LIN {X 0,Y 537.383,Z 578.92,A -85,B 0,C 180,E1 13527.001,E2 13527.001} C_VEL
LIN {X 0,Y 529.562,Z 566.226,A -85,B 0,C 180,E1 13524.901,E2 13524.901} C_VEL
LIN {X 0,Y 521.572,Z 553.811,A -85,B 0,C 180,E1 13522.516,E2 13522.516} C_VEL
LIN {X 0,Y 516.394,Z 546.392,A -85,B 0,C 180,E1 13520.813,E2 13520.813} C_VEL
LIN {X 0,Y 512.056,Z 540.726,A -85,B 0,C 180,E1 13519.269,E2 13519.269} C_VEL
LIN {X 0,Y 508.587,Z 536.104,A -85,B 0,C 180,E1 13517.92,E2 13517.92} C_VEL
LIN {X 0,Y 504.863,Z 531.253,A -85,B 0,C 180,E1 13516.334,E2 13516.334} C_VEL
LIN {X 0,Y 500.708,Z 525.881,A -85,B 0,C 180,E1 13514.337,E2 13514.337} C_VEL
LIN {X 0,Y 497.179,Z 521.35,A -85,B 0,C 180,E1 13512.368,E2 13512.368} C_VEL
LIN {X 0,Y 496.154,Z 520.239,A -85,B 0,C 180,E1 13511.744,E2 13511.744} C_VEL
LIN {X 0,Y 493.12,Z 516.689,A -85,B 0,C 180,E1 13509.63,E2 13509.63} C_VEL
LIN {X 0,Y 492.007,Z 514.619,A -85,B 0,C 180,E1 13508.649,E2 13508.649} C_VEL
LIN {X 0,Y 488.49,Z 511.258,A -85,B 0,C 180,E1 13504.814,E2 13504.814} C_VEL
LIN {X 0,Y 487.575,Z 508.451,A -85,B 0,C 180,E1 13502.586,E2 13502.586} C_VEL
LIN {X 0,Y 487.677,Z 508.543,A -85,B 0,C 180,E1 13496.944,E2 13496.944} C_VEL
LIN {X 0,Y 489.061,Z 512.155,A -85,B 0,C 180,E1 13494.133,E2 13494.133} C_VEL
LIN {X 0,Y 492.312,Z 515.044,A -85,B 0,C 180,E1 13490.885,E2 13490.885} C_VEL
LIN {X 0,Y 494.788,Z 518.967,A -85,B 0,C 180,E1 13488.932,E2 13488.932} C_VEL
LIN {X 0,Y 497.063,Z 521.09,A -85,B 0,C 180,E1 13487.511,E2 13487.511} C_VEL
LIN {X 0,Y 500.333,Z 525.532,A -85,B 0,C 180,E1 13485.652,E2 13485.652} C_VEL
LIN {X 0,Y 501.775,Z 527.195,A -85,B 0,C 180,E1 13484.927,E2 13484.927} C_VEL
LIN {X 0,Y 506.329,Z 533.051,A -85,B 0,C 180,E1 13482.829,E2 13482.829} C_VEL
LIN {X 0,Y 510.668,Z 538.785,A -85,B 0,C 180,E1 13481.062,E2 13481.062} C_VEL
LIN {X 0,Y 515.345,Z 544.978,A -85,B 0,C 180,E1 13479.351,E2 13479.351} C_VEL
LIN {X 0,Y 521.393,Z 553.124,A -85,B 0,C 180,E1 13477.357,E2 13477.357} C_VEL
LIN {X 0,Y 530.749,Z 566.377,A -85,B 0,C 180,E1 13474.622,E2 13474.622} C_VEL
LIN {X 0,Y 537.468,Z 576.651,A -85,B 0,C 180,E1 13472.848,E2 13472.848} C_VEL
LIN {X 0,Y 523.862,Z 798.526,A -85,B 0,C 180,E1 13469.41,E2 13469.41} C_VEL
LIN {X 0,Y 517.892,Z 896.828,A -85,B 0,C 180,E1 13467.872,E2 13467.872} C_VEL
LIN {X 0,Y 515.016,Z 924.398,A -85,B 0,C 180,E1 13467.337,E2 13467.337} C_VEL
LIN {X 0,Y 511.178,Z 950.214,A -85,B 0,C 180,E1 13466.657,E2 13466.657} C_VEL
LIN {X 0,Y 507.419,Z 971.275,A -85,B 0,C 180,E1 13465.969,E2 13465.969} C_VEL
LIN {X 0,Y 503.173,Z 991.991,A -85,B 0,C 180,E1 13465.157,E2 13465.157} C_VEL
LIN {X 0,Y 498.223,Z 1013.275,A -85,B 0,C 180,E1 13464.175,E2 13464.175} C_VEL
LIN {X 0,Y 491.354,Z 1039.557,A -85,B 0,C 180,E1 13462.721,E2 13462.721} C_VEL
LIN {X 0,Y 485.232,Z 1060.389,A -85,B 0,C 180,E1 13461.353,E2 13461.353} C_VEL
LIN {X 0,Y 479.356,Z 1078.967,A -85,B 0,C 180,E1 13459.956,E2 13459.956} C_VEL
LIN {X 0,Y 473.288,Z 1097.052,A -85,B 0,C 180,E1 13458.409,E2 13458.409} C_VEL
LIN {X 0,Y 466.28,Z 1117.027,A -85,B 0,C 180,E1 13456.455,E2 13456.455} C_VEL
LIN {X 0,Y 458.434,Z 1138.201,A -85,B 0,C 180,E1 13454.029,E2 13454.029} C_VEL
LIN {X 0,Y 452.259,Z 1154.399,A -85,B 0,C 180,E1 13451.891,E2 13451.891} C_VEL
LIN {X 0,Y 446.822,Z 1168.494,A -85,B 0,C 180,E1 13449.795,E2 13449.795} C_VEL
LIN {X 0,Y 441.09,Z 1183.448,A -85,B 0,C 180,E1 13447.281,E2 13447.281} C_VEL
LIN {X 0,Y 434.669,Z 1200.398,A -85,B 0,C 180,E1 13443.988,E2 13443.988} C_VEL
LIN {X 0,Y 430.001,Z 1213.2,A -85,B 0,C 180,E1 13441.082,E2 13441.082} C_VEL
LIN {X 0,Y 426.459,Z 1223.501,A -85,B 0,C 180,E1 13438.425,E2 13438.425} C_VEL
LIN {X 0,Y 423.356,Z 1233.296,A -85,B 0,C 180,E1 13435.548,E2 13435.548} C_VEL
LIN {X 0,Y 420.395,Z 1243.93,A -85,B 0,C 180,E1 13431.93,E2 13431.93} C_VEL
LIN {X 0,Y 418.337,Z 1252.385,A -85,B 0,C 180,E1 13428.394,E2 13428.394} C_VEL
LIN {X 0,Y 417.21,Z 1258.312,A -85,B 0,C 180,E1 13425.431,E2 13425.431} C_VEL
LIN {X 0,Y 416.656,Z 1262.093,A -85,B 0,C 180,E1 13423.211,E2 13423.211} C_VEL
LIN {X 0,Y 415.459,Z 1263.67,A -85,B 0,C 180,E1 13422.176,E2 13422.176} C_VEL
LIN {X 0,Y 408.671,Z 1267.583,A -85,B 0,C 180,E1 13419.258,E2 13419.258} C_VEL
LIN {X 0,Y 408.057,Z 1268.429,A -85,B 0,C 180,E1 13418.49,E2 13418.49} C_VEL
LIN {X 0,Y 407.93,Z 1271.067,A -85,B 0,C 180,E1 13414.925,E2 13414.925} C_VEL
LIN {X 0,Y 407.909,Z 1272.244,A -85,B 0,C 180,E1 13411.83,E2 13411.83} C_VEL
LIN {X 0,Y 407.876,Z 1272.395,A -85,B 0,C 180,E1 13409.021,E2 13409.021} C_VEL
LIN {X 0,Y 407.92,Z 1271.653,A -85,B 0,C 180,E1 13406.21,E2 13406.21} C_VEL
LIN {X 0,Y 407.978,Z 1269.903,A -85,B 0,C 180,E1 13403.248,E2 13403.248} C_VEL
LIN {X 0,Y 408.103,Z 1267.313,A -85,B 0,C 180,E1 13400.414,E2 13400.414} C_VEL
LIN {X 0,Y 408.502,Z 1263.796,A -85,B 0,C 180,E1 13397.566,E2 13397.566} C_VEL
LIN {X 0,Y 409.143,Z 1259.33,A -85,B 0,C 180,E1 13394.701,E2 13394.701} C_VEL
LIN {X 0,Y 410.22,Z 1253.882,A -85,B 0,C 180,E1 13391.826,E2 13391.826} C_VEL
LIN {X 0,Y 411.74,Z 1247.416,A -85,B 0,C 180,E1 13388.941,E2 13388.941} C_VEL
LIN {X 0,Y 413.834,Z 1239.881,A -85,B 0,C 180,E1 13386.057,E2 13386.057} C_VEL
LIN {X 0,Y 416.914,Z 1230.158,A -85,B 0,C 180,E1 13382.846,E2 13382.846} C_VEL
LIN {X 0,Y 421.691,Z 1216.502,A -85,B 0,C 180,E1 13379.04,E2 13379.04} C_VEL
LIN {X 0,Y 426.239,Z 1204.343,A -85,B 0,C 180,E1 13376.143,E2 13376.143} C_VEL
LIN {X 0,Y 431.014,Z 1192.094,A -85,B 0,C 180,E1 13373.574,E2 13373.574} C_VEL
LIN {X 0,Y 436.654,Z 1178.048,A -85,B 0,C 180,E1 13370.978,E2 13370.978} C_VEL
LIN {X 0,Y 444.619,Z 1158.26,A -85,B 0,C 180,E1 13367.836,E2 13367.836} C_VEL
LIN {X 0,Y 451.022,Z 1142.083,A -85,B 0,C 180,E1 13365.625,E2 13365.625} C_VEL
LIN {X 0,Y 457.123,Z 1126.351,A -85,B 0,C 180,E1 13363.726,E2 13363.726} C_VEL
LIN {X 0,Y 463.491,Z 1109.375,A -85,B 0,C 180,E1 13361.912,E2 13361.912} C_VEL
LIN {X 0,Y 471.216,Z 1087.969,A -85,B 0,C 180,E1 13359.917,E2 13359.917} C_VEL
LIN {X 0,Y 478.624,Z 1065.488,A -85,B 0,C 180,E1 13358.146,E2 13358.146} C_VEL
LIN {X 0,Y 484.306,Z 1046.983,A -85,B 0,C 180,E1 13356.877,E2 13356.877} C_VEL
LIN {X 0,Y 489.939,Z 1027.141,A -85,B 0,C 180,E1 13355.693,E2 13355.693} C_VEL
LIN {X 0,Y 495.209,Z 1006.776,A -85,B 0,C 180,E1 13354.644,E2 13354.644} C_VEL
LIN {X 0,Y 501.074,Z 981.371,A -85,B 0,C 180,E1 13353.54,E2 13353.54} C_VEL
LIN {X 0,Y 505.952,Z 955.611,A -85,B 0,C 180,E1 13352.647,E2 13352.647} C_VEL
LIN {X 0,Y 509.391,Z 934.091,A -85,B 0,C 180,E1 13352.045,E2 13352.045} C_VEL
LIN {X 0,Y 512.171,Z 912.621,A -85,B 0,C 180,E1 13351.563,E2 13351.563} C_VEL
LIN {X 0,Y 514.439,Z 888.17,A -85,B 0,C 180,E1 13351.127,E2 13351.127} C_VEL
LIN {X 0,Y 528.074,Z 667.756,A -85,B 0,C 180,E1 13347.704,E2 13347.704} C_VEL
LIN {X 0,Y 533.562,Z 581.203,A -85,B 0,C 180,E1 13346.338,E2 13346.338} C_VEL
LIN {X 0,Y 524.924,Z 568.32,A -85,B 0,C 180,E1 13343.937,E2 13343.937} C_VEL
LIN {X 0,Y 517.272,Z 557.54,A -85,B 0,C 180,E1 13341.548,E2 13341.548} C_VEL
LIN {X 0,Y 511.24,Z 549.281,A -85,B 0,C 180,E1 13339.42,E2 13339.42} C_VEL
LIN {X 0,Y 506.838,Z 543.484,A -85,B 0,C 180,E1 13337.687,E2 13337.687} C_VEL
LIN {X 0,Y 503.323,Z 538.833,A -85,B 0,C 180,E1 13336.148,E2 13336.148} C_VEL
LIN {X 0,Y 499.374,Z 533.637,A -85,B 0,C 180,E1 13334.198,E2 13334.198} C_VEL
LIN {X 0,Y 495.757,Z 528.818,A -85,B 0,C 180,E1 13332.108,E2 13332.108} C_VEL
LIN {X 0,Y 492.122,Z 524.788,A -85,B 0,C 180,E1 13329.591,E2 13329.591} C_VEL
LIN {X 0,Y 490.983,Z 522.554,A -85,B 0,C 180,E1 13328.55,E2 13328.55} C_VEL
LIN {X 0,Y 487.467,Z 519.097,A -85,B 0,C 180,E1 13324.471,E2 13324.471} C_VEL
LIN {X 0,Y 486.665,Z 516.418,A -85,B 0,C 180,E1 13322.119,E2 13322.119} C_VEL
LIN {X 0,Y 486.754,Z 516.623,A -85,B 0,C 180,E1 13317.645,E2 13317.645} C_VEL
LIN {X 0,Y 488.538,Z 520.726,A -85,B 0,C 180,E1 13314.008,E2 13314.008} C_VEL
LIN {X 0,Y 491.223,Z 522.944,A -85,B 0,C 180,E1 13311.337,E2 13311.337} C_VEL
LIN {X 0,Y 493.612,Z 526.868,A -85,B 0,C 180,E1 13309.378,E2 13309.378} C_VEL
LIN {X 0,Y 495.917,Z 529.101,A -85,B 0,C 180,E1 13307.896,E2 13307.896} C_VEL
LIN {X 0,Y 499.246,Z 533.532,A -85,B 0,C 180,E1 13305.975,E2 13305.975} C_VEL
LIN {X 0,Y 500.968,Z 535.922,A -85,B 0,C 180,E1 13305.08,E2 13305.08} C_VEL
LIN {X 0,Y 504.775,Z 540.713,A -85,B 0,C 180,E1 13303.308,E2 13303.308} C_VEL
LIN {X 0,Y 508.962,Z 546.319,A -85,B 0,C 180,E1 13301.561,E2 13301.561} C_VEL
LIN {X 0,Y 513.773,Z 552.804,A -85,B 0,C 180,E1 13299.761,E2 13299.761} C_VEL
LIN {X 0,Y 517.708,Z 558.28,A -85,B 0,C 180,E1 13298.412,E2 13298.412} C_VEL
LIN {X 0,Y 526.082,Z 571.313,A -85,B 0,C 180,E1 13295.791,E2 13295.791} C_VEL
LIN {X 0,Y 533.501,Z 583.505,A -85,B 0,C 180,E1 13293.715,E2 13293.715} C_VEL
LIN {X 0,Y 533.493,Z 585.606,A -85,B 0,C 180,E1 13293.655,E2 13293.655} C_VEL
LIN {X 0,Y 519.603,Z 806.043,A -85,B 0,C 180,E1 13290.232,E2 13290.232} C_VEL
LIN {X 0,Y 513.563,Z 902.735,A -85,B 0,C 180,E1 13288.715,E2 13288.715} C_VEL
LIN {X 0,Y 510.594,Z 930.381,A -85,B 0,C 180,E1 13288.183,E2 13288.183} C_VEL
LIN {X 0,Y 506.592,Z 956.342,A -85,B 0,C 180,E1 13287.511,E2 13287.511} C_VEL
LIN {X 0,Y 502.768,Z 977.128,A -85,B 0,C 180,E1 13286.843,E2 13286.843} C_VEL
LIN {X 0,Y 498.39,Z 997.814,A -85,B 0,C 180,E1 13286.045,E2 13286.045} C_VEL
LIN {X 0,Y 493.555,Z 1018.096,A -85,B 0,C 180,E1 13285.124,E2 13285.124} C_VEL
LIN {X 0,Y 487.244,Z 1042.006,A -85,B 0,C 180,E1 13283.844,E2 13283.844} C_VEL
LIN {X 0,Y 480.074,Z 1065.88,A -85,B 0,C 180,E1 13282.313,E2 13282.313} C_VEL
LIN {X 0,Y 473.85,Z 1085.096,A -85,B 0,C 180,E1 13280.881,E2 13280.881} C_VEL
LIN {X 0,Y 467.712,Z 1102.974,A -85,B 0,C 180,E1 13279.361,E2 13279.361} C_VEL
LIN {X 0,Y 460.875,Z 1121.954,A -85,B 0,C 180,E1 13277.523,E2 13277.523} C_VEL
LIN {X 0,Y 452.361,Z 1144.449,A -85,B 0,C 180,E1 13274.982,E2 13274.982} C_VEL
LIN {X 0,Y 445.676,Z 1161.535,A -85,B 0,C 180,E1 13272.732,E2 13272.732} C_VEL
LIN {X 0,Y 439.88,Z 1176.213,A -85,B 0,C 180,E1 13270.542,E2 13270.542} C_VEL
LIN {X 0,Y 434.181,Z 1190.685,A -85,B 0,C 180,E1 13268.104,E2 13268.104} C_VEL
LIN {X 0,Y 427.57,Z 1207.777,A -85,B 0,C 180,E1 13264.786,E2 13264.786} C_VEL
LIN {X 0,Y 422.662,Z 1220.787,A -85,B 0,C 180,E1 13261.834,E2 13261.834} C_VEL
LIN {X 0,Y 418.813,Z 1231.794,A -85,B 0,C 180,E1 13258.983,E2 13258.983} C_VEL
LIN {X 0,Y 415.505,Z 1241.994,A -85,B 0,C 180,E1 13255.969,E2 13255.969} C_VEL
LIN {X 0,Y 412.359,Z 1253.064,A -85,B 0,C 180,E1 13252.138,E2 13252.138} C_VEL
LIN {X 0,Y 410.318,Z 1261.4,A -85,B 0,C 180,E1 13248.611,E2 13248.611} C_VEL
LIN {X 0,Y 409.181,Z 1267.373,A -85,B 0,C 180,E1 13245.588,E2 13245.588} C_VEL
LIN {X 0,Y 408.504,Z 1272.043,A -85,B 0,C 180,E1 13242.721,E2 13242.721} C_VEL
LIN {X 0,Y 408.103,Z 1275.745,A -85,B 0,C 180,E1 13239.871,E2 13239.871} C_VEL
LIN {X 0,Y 407.973,Z 1278.502,A -85,B 0,C 180,E1 13237.035,E2 13237.035} C_VEL
LIN {X 0,Y 407.918,Z 1280.331,A -85,B 0,C 180,E1 13234.213,E2 13234.213} C_VEL
LIN {X 0,Y 407.904,Z 1281.22,A -85,B 0,C 180,E1 13231.541,E2 13231.541} C_VEL
LIN {X 0,Y 407.884,Z 1281.287,A -85,B 0,C 180,E1 13228.872,E2 13228.872} C_VEL
LIN {X 0,Y 407.918,Z 1280.464,A -85,B 0,C 180,E1 13226.061,E2 13226.061} C_VEL
LIN {X 0,Y 407.964,Z 1278.724,A -85,B 0,C 180,E1 13223.24,E2 13223.24} C_VEL
LIN {X 0,Y 408.077,Z 1276.057,A -85,B 0,C 180,E1 13220.405,E2 13220.405} C_VEL
LIN {X 0,Y 408.461,Z 1272.448,A -85,B 0,C 180,E1 13217.556,E2 13217.556} C_VEL
LIN {X 0,Y 409.133,Z 1267.614,A -85,B 0,C 180,E1 13214.547,E2 13214.547} C_VEL
LIN {X 0,Y 410.193,Z 1261.991,A -85,B 0,C 180,E1 13211.669,E2 13211.669} C_VEL
LIN {X 0,Y 411.824,Z 1254.979,A -85,B 0,C 180,E1 13208.639,E2 13208.639} C_VEL
LIN {X 0,Y 414.433,Z 1245.558,A -85,B 0,C 180,E1 13205.175,E2 13205.175} C_VEL
LIN {X 0,Y 418.291,Z 1233.317,A -85,B 0,C 180,E1 13201.437,E2 13201.437} C_VEL
LIN {X 0,Y 422.06,Z 1222.479,A -85,B 0,C 180,E1 13198.585,E2 13198.585} C_VEL
LIN {X 0,Y 426.369,Z 1210.799,A -85,B 0,C 180,E1 13195.877,E2 13195.877} C_VEL
LIN {X 0,Y 431.872,Z 1196.608,A -85,B 0,C 180,E1 13192.987,E2 13192.987} C_VEL
LIN {X 0,Y 438.91,Z 1178.681,A -85,B 0,C 180,E1 13189.854,E2 13189.854} C_VEL
LIN {X 0,Y 444.971,Z 1163.303,A -85,B 0,C 180,E1 13187.524,E2 13187.524} C_VEL
LIN {X 0,Y 451.05,Z 1147.752,A -85,B 0,C 180,E1 13185.441,E2 13185.441} C_VEL
LIN {X 0,Y 457.429,Z 1131.105,A -85,B 0,C 180,E1 13183.469,E2 13183.469} C_VEL
LIN {X 0,Y 465.426,Z 1109.512,A -85,B 0,C 180,E1 13181.241,E2 13181.241} C_VEL
LIN {X 0,Y 472.738,Z 1088.316,A -85,B 0,C 180,E1 13179.386,E2 13179.386} C_VEL
LIN {X 0,Y 478.815,Z 1069.74,A -85,B 0,C 180,E1 13177.969,E2 13177.969} C_VEL
LIN {X 0,Y 484.294,Z 1051.797,A -85,B 0,C 180,E1 13176.765,E2 13176.765} C_VEL
LIN {X 0,Y 489.677,Z 1032.685,A -85,B 0,C 180,E1 13175.638,E2 13175.638} C_VEL
LIN {X 0,Y 495.065,Z 1011.807,A -85,B 0,C 180,E1 13174.579,E2 13174.579} C_VEL
LIN {X 0,Y 501.236,Z 984.578,A -85,B 0,C 180,E1 13173.43,E2 13173.43} C_VEL
LIN {X 0,Y 505.715,Z 961.031,A -85,B 0,C 180,E1 13172.634,E2 13172.634} C_VEL
LIN {X 0,Y 509.157,Z 939.541,A -85,B 0,C 180,E1 13172.041,E2 13172.041} C_VEL
LIN {X 0,Y 512.025,Z 917.551,A -85,B 0,C 180,E1 13171.561,E2 13171.561} C_VEL
LIN {X 0,Y 514.484,Z 890.024,A -85,B 0,C 180,E1 13171.076,E2 13171.076} C_VEL
LIN {X 0,Y 528.167,Z 667.075,A -85,B 0,C 180,E1 13167.618,E2 13167.618} C_VEL
LIN {X 0,Y 533.496,Z 583.585,A -85,B 0,C 180,E1 13166.312,E2 13166.312} C_VEL
LIN {X 0,Y 526.499,Z 572.116,A -85,B 0,C 180,E1 13164.367,E2 13164.367} C_VEL
LIN {X 0,Y 519.099,Z 560.49,A -85,B 0,C 180,E1 13162.092,E2 13162.092} C_VEL
LIN {X 0,Y 514.331,Z 553.562,A -85,B 0,C 180,E1 13160.483,E2 13160.483} C_VEL
LIN {X 0,Y 510.071,Z 547.908,A -85,B 0,C 180,E1 13158.931,E2 13158.931} C_VEL
LIN {X 0,Y 506.803,Z 543.491,A -85,B 0,C 180,E1 13157.629,E2 13157.629} C_VEL
LIN {X 0,Y 503.27,Z 538.812,A -85,B 0,C 180,E1 13156.091,E2 13156.091} C_VEL
LIN {X 0,Y 499.187,Z 533.475,A -85,B 0,C 180,E1 13154.086,E2 13154.086} C_VEL
LIN {X 0,Y 495.654,Z 528.732,A -85,B 0,C 180,E1 13152.052,E2 13152.052} C_VEL
LIN {X 0,Y 492.061,Z 524.745,A -85,B 0,C 180,E1 13149.592,E2 13149.592} C_VEL
LIN {X 0,Y 490.898,Z 522.51,A -85,B 0,C 180,E1 13148.551,E2 13148.551} C_VEL
LIN {X 0,Y 487.441,Z 519.137,A -85,B 0,C 180,E1 13144.707,E2 13144.707} C_VEL
LIN {X 0,Y 486.556,Z 516.384,A -85,B 0,C 180,E1 13142.473,E2 13142.473} C_VEL
LIN {X 0,Y 486.687,Z 516.619,A -85,B 0,C 180,E1 13136.938,E2 13136.938} C_VEL
LIN {X 0,Y 488.172,Z 520.264,A -85,B 0,C 180,E1 13134.004,E2 13134.004} C_VEL
LIN {X 0,Y 491.129,Z 522.882,A -85,B 0,C 180,E1 13131.04,E2 13131.04} C_VEL
LIN {X 0,Y 493.647,Z 526.856,A -85,B 0,C 180,E1 13129.024,E2 13129.024} C_VEL
LIN {X 0,Y 495.799,Z 528.961,A -85,B 0,C 180,E1 13127.656,E2 13127.656} C_VEL
LIN {X 0,Y 499.147,Z 533.437,A -85,B 0,C 180,E1 13125.736,E2 13125.736} C_VEL
LIN {X 0,Y 500.56,Z 535.265,A -85,B 0,C 180,E1 13125.008,E2 13125.008} C_VEL
LIN {X 0,Y 504.836,Z 540.791,A -85,B 0,C 180,E1 13123.014,E2 13123.014} C_VEL
LIN {X 0,Y 509.055,Z 546.447,A -85,B 0,C 180,E1 13121.268,E2 13121.268} C_VEL
LIN {X 0,Y 515.524,Z 555.003,A -85,B 0,C 180,E1 13118.913,E2 13118.913} C_VEL
LIN {X 0,Y 523.859,Z 566.89,A -85,B 0,C 180,E1 13116.251,E2 13116.251} C_VEL
LIN {X 0,Y 531.87,Z 578.695,A -85,B 0,C 180,E1 13113.992,E2 13113.992} C_VEL
LIN {X 0,Y 533.543,Z 581.496,A -85,B 0,C 180,E1 13113.541,E2 13113.541} C_VEL
LIN {X 0,Y 519.553,Z 803.097,A -85,B 0,C 180,E1 13110.102,E2 13110.102} C_VEL
LIN {X 0,Y 513.663,Z 897.047,A -85,B 0,C 180,E1 13108.628,E2 13108.628} C_VEL
LIN {X 0,Y 510.691,Z 924.741,A -85,B 0,C 180,E1 13108.09,E2 13108.09} C_VEL
LIN {X 0,Y 506.791,Z 950.352,A -85,B 0,C 180,E1 13107.416,E2 13107.416} C_VEL
LIN {X 0,Y 502.853,Z 971.844,A -85,B 0,C 180,E1 13106.714,E2 13106.714} C_VEL
LIN {X 0,Y 498.591,Z 992.088,A -85,B 0,C 180,E1 13105.92,E2 13105.92} C_VEL
LIN {X 0,Y 493.51,Z 1013.372,A -85,B 0,C 180,E1 13104.94,E2 13104.94} C_VEL
LIN {X 0,Y 486.455,Z 1039.652,A -85,B 0,C 180,E1 13103.485,E2 13103.485} C_VEL
LIN {X 0,Y 480.153,Z 1060.485,A -85,B 0,C 180,E1 13102.117,E2 13102.117} C_VEL
LIN {X 0,Y 474.097,Z 1079.062,A -85,B 0,C 180,E1 13100.718,E2 13100.718} C_VEL
LIN {X 0,Y 467.781,Z 1097.323,A -85,B 0,C 180,E1 13099.15,E2 13099.15} C_VEL
LIN {X 0,Y 460.174,Z 1118.334,A -85,B 0,C 180,E1 13097.078,E2 13097.078} C_VEL
LIN {X 0,Y 452.419,Z 1138.439,A -85,B 0,C 180,E1 13094.744,E2 13094.744} C_VEL
LIN {X 0,Y 446.069,Z 1154.494,A -85,B 0,C 180,E1 13092.608,E2 13092.608} C_VEL
LIN {X 0,Y 440.4,Z 1168.641,A -85,B 0,C 180,E1 13090.484,E2 13090.484} C_VEL
LIN {X 0,Y 434.685,Z 1182.926,A -85,B 0,C 180,E1 13088.061,E2 13088.061} C_VEL
LIN {X 0,Y 428.273,Z 1199.231,A -85,B 0,C 180,E1 13084.893,E2 13084.893} C_VEL
LIN {X 0,Y 423.044,Z 1212.725,A -85,B 0,C 180,E1 13081.811,E2 13081.811} C_VEL
LIN {X 0,Y 419.133,Z 1223.594,A -85,B 0,C 180,E1 13078.968,E2 13078.968} C_VEL
LIN {X 0,Y 415.913,Z 1233.199,A -85,B 0,C 180,E1 13076.104,E2 13076.104} C_VEL
LIN {X 0,Y 412.92,Z 1243.226,A -85,B 0,C 180,E1 13072.648,E2 13072.648} C_VEL
LIN {X 0,Y 410.596,Z 1252.177,A -85,B 0,C 180,E1 13068.901,E2 13068.901} C_VEL
LIN {X 0,Y 409.328,Z 1258.402,A -85,B 0,C 180,E1 13065.736,E2 13065.736} C_VEL
LIN {X 0,Y 408.563,Z 1263.247,A -85,B 0,C 180,E1 13062.728,E2 13062.728} C_VEL
LIN {X 0,Y 408.136,Z 1266.886,A -85,B 0,C 180,E1 13059.878,E2 13059.878} C_VEL
LIN {X 0,Y 408.057,Z 1268.429,A -85,B 0,C 180,E1 13058.49,E2 13058.49} C_VEL
LIN {X 0,Y 406.973,Z 1269.486,A -85,B 0,C 180,E1 13057.42,E2 13057.42} C_VEL
LIN {X 0,Y 400.455,Z 1271.449,A -85,B 0,C 180,E1 13054.387,E2 13054.387} C_VEL
LIN {X 0,Y 399.92,Z 1271.826,A -85,B 0,C 180,E1 13053.592,E2 13053.592} C_VEL
LIN {X 0,Y 399.905,Z 1272.624,A -85,B 0,C 180,E1 13050.004,E2 13050.004} C_VEL
LIN {X 0,Y 399.919,Z 1271.875,A -85,B 0,C 180,E1 13046.421,E2 13046.421} C_VEL
LIN {X 0,Y 399.98,Z 1270.103,A -85,B 0,C 180,E1 13043.257,E2 13043.257} C_VEL
LIN {X 0,Y 400.111,Z 1267.559,A -85,B 0,C 180,E1 13040.366,E2 13040.366} C_VEL
LIN {X 0,Y 400.551,Z 1263.884,A -85,B 0,C 180,E1 13037.315,E2 13037.315} C_VEL
LIN {X 0,Y 401.309,Z 1259.166,A -85,B 0,C 180,E1 13034.247,E2 13034.247} C_VEL
LIN {X 0,Y 402.54,Z 1253.347,A -85,B 0,C 180,E1 13031.154,E2 13031.154} C_VEL
LIN {X 0,Y 404.442,Z 1246.105,A -85,B 0,C 180,E1 13027.933,E2 13027.933} C_VEL
LIN {X 0,Y 407.753,Z 1235.407,A -85,B 0,C 180,E1 13023.969,E2 13023.969} C_VEL
LIN {X 0,Y 411.534,Z 1224.522,A -85,B 0,C 180,E1 13020.614,E2 13020.614} C_VEL
LIN {X 0,Y 415.366,Z 1214.315,A -85,B 0,C 180,E1 13017.866,E2 13017.866} C_VEL
LIN {X 0,Y 419.922,Z 1202.875,A -85,B 0,C 180,E1 13015.154,E2 13015.154} C_VEL
LIN {X 0,Y 426.116,Z 1188.005,A -85,B 0,C 180,E1 13012.071,E2 13012.071} C_VEL
LIN {X 0,Y 433.208,Z 1170.885,A -85,B 0,C 180,E1 13009.05,E2 13009.05} C_VEL
LIN {X 0,Y 439.536,Z 1155.677,A -85,B 0,C 180,E1 13006.716,E2 13006.716} C_VEL
LIN {X 0,Y 445.909,Z 1140.152,A -85,B 0,C 180,E1 13004.614,E2 13004.614} C_VEL
LIN {X 0,Y 452.992,Z 1122.485,A -85,B 0,C 180,E1 13002.512,E2 13002.512} C_VEL
LIN {X 0,Y 461.771,Z 1099.367,A -85,B 0,C 180,E1 13000.158,E2 13000.158} C_VEL
LIN {X 0,Y 468.506,Z 1080.548,A -85,B 0,C 180,E1 12998.52,E2 12998.52} C_VEL
LIN {X 0,Y 474.646,Z 1062.336,A -85,B 0,C 180,E1 12997.132,E2 12997.132} C_VEL
LIN {X 0,Y 480.272,Z 1044.372,A -85,B 0,C 180,E1 12995.927,E2 12995.927} C_VEL
LIN {X 0,Y 486.362,Z 1023.213,A -85,B 0,C 180,E1 12994.69,E2 12994.69} C_VEL
LIN {X 0,Y 493.259,Z 996.204,A -85,B 0,C 180,E1 12993.377,E2 12993.377} C_VEL
LIN {X 0,Y 498.116,Z 974.04,A -85,B 0,C 180,E1 12992.49,E2 12992.49} C_VEL
LIN {X 0,Y 502.157,Z 952.827,A -85,B 0,C 180,E1 12991.787,E2 12991.787} C_VEL
LIN {X 0,Y 505.55,Z 931.576,A -85,B 0,C 180,E1 12991.207,E2 12991.207} C_VEL
LIN {X 0,Y 508.778,Z 906.365,A -85,B 0,C 180,E1 12990.668,E2 12990.668} C_VEL
LIN {X 0,Y 511.592,Z 868.962,A -85,B 0,C 180,E1 12990.051,E2 12990.051} C_VEL
LIN {X 0,Y 525.613,Z 649.177,A -85,B 0,C 180,E1 12986.637,E2 12986.637} C_VEL
LIN {X 0,Y 529.741,Z 586.102,A -85,B 0,C 180,E1 12985.64,E2 12985.64} C_VEL
LIN {X 0,Y 522.109,Z 574.631,A -85,B 0,C 180,E1 12983.445,E2 12983.445} C_VEL
LIN {X 0,Y 515.027,Z 564.467,A -85,B 0,C 180,E1 12981.168,E2 12981.168} C_VEL
LIN {X 0,Y 508.97,Z 556.133,A -85,B 0,C 180,E1 12978.974,E2 12978.974} C_VEL
LIN {X 0,Y 505.072,Z 550.871,A -85,B 0,C 180,E1 12977.394,E2 12977.394} C_VEL
LIN {X 0,Y 501.743,Z 546.391,A -85,B 0,C 180,E1 12975.903,E2 12975.903} C_VEL
LIN {X 0,Y 497.864,Z 541.232,A -85,B 0,C 180,E1 12973.946,E2 12973.946} C_VEL
LIN {X 0,Y 494.058,Z 536.136,A -85,B 0,C 180,E1 12971.676,E2 12971.676} C_VEL
LIN {X 0,Y 490.93,Z 532.597,A -85,B 0,C 180,E1 12969.437,E2 12969.437} C_VEL
LIN {X 0,Y 489.741,Z 530.38,A -85,B 0,C 180,E1 12968.335,E2 12968.335} C_VEL
LIN {X 0,Y 486.427,Z 526.977,A -85,B 0,C 180,E1 12964.362,E2 12964.362} C_VEL
LIN {X 0,Y 485.656,Z 524.353,A -85,B 0,C 180,E1 12962.006,E2 12962.006} C_VEL
LIN {X 0,Y 485.746,Z 524.507,A -85,B 0,C 180,E1 12957.759,E2 12957.759} C_VEL
LIN {X 0,Y 487.529,Z 528.665,A -85,B 0,C 180,E1 12954.04,E2 12954.04} C_VEL
LIN {X 0,Y 490.047,Z 530.778,A -85,B 0,C 180,E1 12951.493,E2 12951.493} C_VEL
LIN {X 0,Y 492.476,Z 534.756,A -85,B 0,C 180,E1 12949.471,E2 12949.471} C_VEL
LIN {X 0,Y 494.575,Z 536.799,A -85,B 0,C 180,E1 12948.099,E2 12948.099} C_VEL
LIN {X 0,Y 498.062,Z 541.431,A -85,B 0,C 180,E1 12946.06,E2 12946.06} C_VEL
LIN {X 0,Y 503.292,Z 548.448,A -85,B 0,C 180,E1 12943.495,E2 12943.495} C_VEL
LIN {X 0,Y 507.427,Z 554.073,A -85,B 0,C 180,E1 12941.741,E2 12941.741} C_VEL
LIN {X 0,Y 513.78,Z 562.635,A -85,B 0,C 180,E1 12939.375,E2 12939.375} C_VEL
LIN {X 0,Y 521.313,Z 574.374,A -85,B 0,C 180,E1 12936.876,E2 12936.876} C_VEL
LIN {X 0,Y 528.597,Z 586.377,A -85,B 0,C 180,E1 12934.721,E2 12934.721} C_VEL
LIN {X 0,Y 529.774,Z 588.511,A -85,B 0,C 180,E1 12934.388,E2 12934.388} C_VEL
LIN {X 0,Y 515.437,Z 809.52,A -85,B 0,C 180,E1 12930.952,E2 12930.952} C_VEL
LIN {X 0,Y 509.425,Z 902.796,A -85,B 0,C 180,E1 12929.485,E2 12929.485} C_VEL
LIN {X 0,Y 506.36,Z 930.566,A -85,B 0,C 180,E1 12928.95,E2 12928.95} C_VEL
LIN {X 0,Y 502.281,Z 956.381,A -85,B 0,C 180,E1 12928.285,E2 12928.285} C_VEL
LIN {X 0,Y 498.282,Z 977.574,A -85,B 0,C 180,E1 12927.603,E2 12927.603} C_VEL
LIN {X 0,Y 493.901,Z 997.732,A -85,B 0,C 180,E1 12926.827,E2 12926.827} C_VEL
LIN {X 0,Y 488.942,Z 1018.013,A -85,B 0,C 180,E1 12925.907,E2 12925.907} C_VEL
LIN {X 0,Y 482.454,Z 1041.922,A -85,B 0,C 180,E1 12924.63,E2 12924.63} C_VEL
LIN {X 0,Y 475.085,Z 1065.794,A -85,B 0,C 180,E1 12923.099,E2 12923.099} C_VEL
LIN {X 0,Y 468.545,Z 1085.403,A -85,B 0,C 180,E1 12921.633,E2 12921.633} C_VEL
LIN {X 0,Y 462.115,Z 1103.557,A -85,B 0,C 180,E1 12920.08,E2 12920.08} C_VEL
LIN {X 0,Y 454.845,Z 1123.088,A -85,B 0,C 180,E1 12918.17,E2 12918.17} C_VEL
LIN {X 0,Y 446.122,Z 1145.238,A -85,B 0,C 180,E1 12915.63,E2 12915.63} C_VEL
LIN {X 0,Y 439.547,Z 1161.442,A -85,B 0,C 180,E1 12913.475,E2 12913.475} C_VEL
LIN {X 0,Y 433.437,Z 1176.331,A -85,B 0,C 180,E1 12911.232,E2 12911.232} C_VEL
LIN {X 0,Y 427.276,Z 1191.37,A -85,B 0,C 180,E1 12908.662,E2 12908.662} C_VEL
LIN {X 0,Y 420.151,Z 1208.964,A -85,B 0,C 180,E1 12905.157,E2 12905.157} C_VEL
LIN {X 0,Y 415.313,Z 1221.274,A -85,B 0,C 180,E1 12902.302,E2 12902.302} C_VEL
LIN {X 0,Y 411.487,Z 1231.703,A -85,B 0,C 180,E1 12899.55,E2 12899.55} C_VEL
LIN {X 0,Y 407.997,Z 1241.904,A -85,B 0,C 180,E1 12896.483,E2 12896.483} C_VEL
LIN {X 0,Y 404.723,Z 1252.776,A -85,B 0,C 180,E1 12892.663,E2 12892.663} C_VEL
LIN {X 0,Y 402.499,Z 1261.31,A -85,B 0,C 180,E1 12888.986,E2 12888.986} C_VEL
LIN {X 0,Y 401.285,Z 1267.313,A -85,B 0,C 180,E1 12885.886,E2 12885.886} C_VEL
LIN {X 0,Y 400.524,Z 1272.163,A -85,B 0,C 180,E1 12882.832,E2 12882.832} C_VEL
LIN {X 0,Y 400.109,Z 1275.818,A -85,B 0,C 180,E1 12879.925,E2 12879.925} C_VEL
LIN {X 0,Y 399.981,Z 1278.414,A -85,B 0,C 180,E1 12877.176,E2 12877.176} C_VEL
LIN {X 0,Y 399.919,Z 1280.244,A -85,B 0,C 180,E1 12874.297,E2 12874.297} C_VEL
LIN {X 0,Y 399.905,Z 1281.133,A -85,B 0,C 180,E1 12871.572,E2 12871.572} C_VEL
LIN {X 0,Y 399.887,Z 1281.2,A -85,B 0,C 180,E1 12868.85,E2 12868.85} C_VEL
LIN {X 0,Y 399.918,Z 1280.377,A -85,B 0,C 180,E1 12865.982,E2 12865.982} C_VEL
LIN {X 0,Y 399.969,Z 1278.636,A -85,B 0,C 180,E1 12863.104,E2 12863.104} C_VEL
LIN {X 0,Y 400.094,Z 1275.968,A -85,B 0,C 180,E1 12860.212,E2 12860.212} C_VEL
LIN {X 0,Y 400.502,Z 1272.358,A -85,B 0,C 180,E1 12857.305,E2 12857.305} C_VEL
LIN {X 0,Y 401.241,Z 1267.524,A -85,B 0,C 180,E1 12854.235,E2 12854.235} C_VEL
LIN {X 0,Y 402.401,Z 1261.719,A -85,B 0,C 180,E1 12851.212,E2 12851.212} C_VEL
LIN {X 0,Y 404.31,Z 1254.174,A -85,B 0,C 180,E1 12847.916,E2 12847.916} C_VEL
LIN {X 0,Y 407.715,Z 1242.796,A -85,B 0,C 180,E1 12843.801,E2 12843.801} C_VEL
LIN {X 0,Y 411.313,Z 1232.187,A -85,B 0,C 180,E1 12840.587,E2 12840.587} C_VEL
LIN {X 0,Y 415.104,Z 1221.808,A -85,B 0,C 180,E1 12837.834,E2 12837.834} C_VEL
LIN {X 0,Y 419.826,Z 1209.727,A -85,B 0,C 180,E1 12835.015,E2 12835.015} C_VEL
LIN {X 0,Y 426.39,Z 1193.62,A -85,B 0,C 180,E1 12831.748,E2 12831.748} C_VEL
LIN {X 0,Y 433.191,Z 1176.887,A -85,B 0,C 180,E1 12828.862,E2 12828.862} C_VEL
LIN {X 0,Y 439.368,Z 1161.812,A -85,B 0,C 180,E1 12826.583,E2 12826.583} C_VEL
LIN {X 0,Y 445.728,Z 1146.13,A -85,B 0,C 180,E1 12824.489,E2 12824.489} C_VEL
LIN {X 0,Y 453.961,Z 1125.385,A -85,B 0,C 180,E1 12822.072,E2 12822.072} C_VEL
LIN {X 0,Y 461.614,Z 1104.813,A -85,B 0,C 180,E1 12820.04,E2 12820.04} C_VEL
LIN {X 0,Y 468.338,Z 1085.849,A -85,B 0,C 180,E1 12818.41,E2 12818.41} C_VEL
LIN {X 0,Y 474.836,Z 1066.391,A -85,B 0,C 180,E1 12816.95,E2 12816.95} C_VEL
LIN {X 0,Y 482.2,Z 1042.657,A -85,B 0,C 180,E1 12815.418,E2 12815.418} C_VEL
LIN {X 0,Y 488.671,Z 1018.838,A -85,B 0,C 180,E1 12814.139,E2 12814.139} C_VEL
LIN {X 0,Y 493.785,Z 997.95,A -85,B 0,C 180,E1 12813.188,E2 12813.188} C_VEL
LIN {X 0,Y 498.219,Z 977.544,A -85,B 0,C 180,E1 12812.402,E2 12812.402} C_VEL
LIN {X 0,Y 502.237,Z 956.222,A -85,B 0,C 180,E1 12811.716,E2 12811.716} C_VEL
LIN {X 0,Y 506.418,Z 929.675,A -85,B 0,C 180,E1 12811.034,E2 12811.034} C_VEL
LIN {X 0,Y 509.388,Z 902.291,A -85,B 0,C 180,E1 12810.512,E2 12810.512} C_VEL
LIN {X 0,Y 517.283,Z 778.951,A -85,B 0,C 180,E1 12808.58,E2 12808.58} C_VEL
LIN {X 0,Y 529.683,Z 588.277,A -85,B 0,C 180,E1 12805.613,E2 12805.613} C_VEL
LIN {X 0,Y 522.38,Z 576.169,A -85,B 0,C 180,E1 12803.492,E2 12803.492} C_VEL
LIN {X 0,Y 514.336,Z 563.548,A -85,B 0,C 180,E1 12800.87,E2 12800.87} C_VEL
LIN {X 0,Y 508.665,Z 555.818,A -85,B 0,C 180,E1 12798.807,E2 12798.807} C_VEL
LIN {X 0,Y 505.032,Z 550.877,A -85,B 0,C 180,E1 12797.336,E2 12797.336} C_VEL
LIN {X 0,Y 501.686,Z 546.369,A -85,B 0,C 180,E1 12795.846,E2 12795.846} C_VEL
LIN {X 0,Y 497.783,Z 541.171,A -85,B 0,C 180,E1 12793.889,E2 12793.889} C_VEL
LIN {X 0,Y 493.852,Z 535.996,A -85,B 0,C 180,E1 12791.563,E2 12791.563} C_VEL
LIN {X 0,Y 490.797,Z 532.433,A -85,B 0,C 180,E1 12789.38,E2 12789.38} C_VEL
LIN {X 0,Y 489.651,Z 530.331,A -85,B 0,C 180,E1 12788.336,E2 12788.336} C_VEL
LIN {X 0,Y 486.331,Z 526.87,A -85,B 0,C 180,E1 12784.481,E2 12784.481} C_VEL
LIN {X 0,Y 485.582,Z 524.325,A -85,B 0,C 180,E1 12782.478,E2 12782.478} C_VEL
LIN {X 0,Y 485.669,Z 524.51,A -85,B 0,C 180,E1 12777.05,E2 12777.05} C_VEL
LIN {X 0,Y 487.108,Z 528.143,A -85,B 0,C 180,E1 12774.109,E2 12774.109} C_VEL
LIN {X 0,Y 489.949,Z 530.716,A -85,B 0,C 180,E1 12771.196,E2 12771.196} C_VEL
LIN {X 0,Y 492.509,Z 534.744,A -85,B 0,C 180,E1 12769.117,E2 12769.117} C_VEL
LIN {X 0,Y 494.539,Z 536.823,A -85,B 0,C 180,E1 12767.802,E2 12767.802} C_VEL
LIN {X 0,Y 497.963,Z 541.338,A -85,B 0,C 180,E1 12765.82,E2 12765.82} C_VEL
LIN {X 0,Y 503.228,Z 548.341,A -85,B 0,C 180,E1 12763.255,E2 12763.255} C_VEL
LIN {X 0,Y 507.382,Z 554.005,A -85,B 0,C 180,E1 12761.501,E2 12761.501} C_VEL
LIN {X 0,Y 513.61,Z 562.383,A -85,B 0,C 180,E1 12759.189,E2 12759.189} C_VEL
LIN {X 0,Y 522.175,Z 574.76,A -85,B 0,C 180,E1 12756.409,E2 12756.409} C_VEL
LIN {X 0,Y 529.711,Z 586.127,A -85,B 0,C 180,E1 12754.248,E2 12754.248} C_VEL
LIN {X 0,Y 515.388,Z 806.61,A -85,B 0,C 180,E1 12750.822,E2 12750.822} C_VEL
LIN {X 0,Y 509.534,Z 897.158,A -85,B 0,C 180,E1 12749.398,E2 12749.398} C_VEL
LIN {X 0,Y 506.475,Z 924.963,A -85,B 0,C 180,E1 12748.858,E2 12748.858} C_VEL
LIN {X 0,Y 502.502,Z 950.452,A -85,B 0,C 180,E1 12748.189,E2 12748.189} C_VEL
LIN {X 0,Y 498.531,Z 971.636,A -85,B 0,C 180,E1 12747.501,E2 12747.501} C_VEL
LIN {X 0,Y 494.099,Z 992.186,A -85,B 0,C 180,E1 12746.698,E2 12746.698} C_VEL
LIN {X 0,Y 488.889,Z 1013.469,A -85,B 0,C 180,E1 12745.72,E2 12745.72} C_VEL
LIN {X 0,Y 481.644,Z 1039.748,A -85,B 0,C 180,E1 12744.266,E2 12744.266} C_VEL
LIN {X 0,Y 475.16,Z 1060.58,A -85,B 0,C 180,E1 12742.898,E2 12742.898} C_VEL
LIN {X 0,Y 468.888,Z 1079.272,A -85,B 0,C 180,E1 12741.488,E2 12741.488} C_VEL
LIN {X 0,Y 462.486,Z 1097.242,A -85,B 0,C 180,E1 12739.94,E2 12739.94} C_VEL
LIN {X 0,Y 455.01,Z 1117.217,A -85,B 0,C 180,E1 12737.969,E2 12737.969} C_VEL
LIN {X 0,Y 446.562,Z 1138.47,A -85,B 0,C 180,E1 12735.506,E2 12735.506} C_VEL
LIN {X 0,Y 439.928,Z 1154.641,A -85,B 0,C 180,E1 12733.338,E2 12733.338} C_VEL
LIN {X 0,Y 433.741,Z 1169.524,A -85,B 0,C 180,E1 12731.074,E2 12731.074} C_VEL
LIN {X 0,Y 427.199,Z 1185.318,A -85,B 0,C 180,E1 12728.337,E2 12728.337} C_VEL
LIN {X 0,Y 420.344,Z 1201.848,A -85,B 0,C 180,E1 12724.982,E2 12724.982} C_VEL
LIN {X 0,Y 415.498,Z 1213.957,A -85,B 0,C 180,E1 12722.132,E2 12722.132} C_VEL
LIN {X 0,Y 411.462,Z 1224.709,A -85,B 0,C 180,E1 12719.242,E2 12719.242} C_VEL
LIN {X 0,Y 407.555,Z 1236.022,A -85,B 0,C 180,E1 12715.741,E2 12715.741} C_VEL
LIN {X 0,Y 404.404,Z 1246.221,A -85,B 0,C 180,E1 12711.926,E2 12711.926} C_VEL
LIN {X 0,Y 402.573,Z 1253.169,A -85,B 0,C 180,E1 12708.841,E2 12708.841} C_VEL
LIN {X 0,Y 401.398,Z 1258.745,A -85,B 0,C 180,E1 12705.907,E2 12705.907} C_VEL
LIN {X 0,Y 400.59,Z 1263.541,A -85,B 0,C 180,E1 12702.839,E2 12702.839} C_VEL
LIN {X 0,Y 400.147,Z 1267.133,A -85,B 0,C 180,E1 12699.932,E2 12699.932} C_VEL
LIN {X 0,Y 399.992,Z 1269.799,A -85,B 0,C 180,E1 12697.04,E2 12697.04} C_VEL
LIN {X 0,Y 399.923,Z 1271.559,A -85,B 0,C 180,E1 12694.162,E2 12694.162} C_VEL
LIN {X 0,Y 399.92,Z 1271.826,A -85,B 0,C 180,E1 12693.592,E2 12693.592} C_VEL
LIN {X 0,Y 399.036,Z 1272.245,A -85,B 0,C 180,E1 12692.568,E2 12692.568} C_VEL
LIN {X 0,Y 394.951,Z 1272.62,A -85,B 0,C 180,E1 12690.721,E2 12690.721} C_VEL
LIN {X 0,Y 392.223,Z 1272.62,A -85,B 0,C 180,E1 12689.219,E2 12689.219} C_VEL
LIN {X 0,Y 391.898,Z 1272.506,A -85,B 0,C 180,E1 12688.567,E2 12688.567} C_VEL
LIN {X 0,Y 391.926,Z 1271.693,A -85,B 0,C 180,E1 12685.762,E2 12685.762} C_VEL
LIN {X 0,Y 391.997,Z 1269.965,A -85,B 0,C 180,E1 12682.825,E2 12682.825} C_VEL
LIN {X 0,Y 392.166,Z 1267.33,A -85,B 0,C 180,E1 12679.872,E2 12679.872} C_VEL
LIN {X 0,Y 392.635,Z 1263.768,A -85,B 0,C 180,E1 12676.905,E2 12676.905} C_VEL
LIN {X 0,Y 393.489,Z 1259.003,A -85,B 0,C 180,E1 12673.774,E2 12673.774} C_VEL
LIN {X 0,Y 394.818,Z 1253.16,A -85,B 0,C 180,E1 12670.63,E2 12670.63} C_VEL
LIN {X 0,Y 397.103,Z 1245.145,A -85,B 0,C 180,E1 12667.034,E2 12667.034} C_VEL
LIN {X 0,Y 400.58,Z 1234.586,A -85,B 0,C 180,E1 12663.147,E2 12663.147} C_VEL
LIN {X 0,Y 404.396,Z 1224.255,A -85,B 0,C 180,E1 12659.928,E2 12659.928} C_VEL
LIN {X 0,Y 408.529,Z 1213.815,A -85,B 0,C 180,E1 12657.088,E2 12657.088} C_VEL
LIN {X 0,Y 413.629,Z 1201.703,A -85,B 0,C 180,E1 12654.204,E2 12654.204} C_VEL
LIN {X 0,Y 421.107,Z 1184.354,A -85,B 0,C 180,E1 12650.664,E2 12650.664} C_VEL
LIN {X 0,Y 427.632,Z 1169.292,A -85,B 0,C 180,E1 12648.039,E2 12648.039} C_VEL
LIN {X 0,Y 434.102,Z 1154.318,A -85,B 0,C 180,E1 12645.748,E2 12645.748} C_VEL
LIN {X 0,Y 441.353,Z 1137.283,A -85,B 0,C 180,E1 12643.461,E2 12643.461} C_VEL
LIN {X 0,Y 450.212,Z 1115.607,A -85,B 0,C 180,E1 12640.973,E2 12640.973} C_VEL
LIN {X 0,Y 457.482,Z 1096.792,A -85,B 0,C 180,E1 12639.122,E2 12639.122} C_VEL
LIN {X 0,Y 464.361,Z 1077.992,A -85,B 0,C 180,E1 12637.509,E2 12637.509} C_VEL
LIN {X 0,Y 471.918,Z 1055.946,A -85,B 0,C 180,E1 12635.872,E2 12635.872} C_VEL
LIN {X 0,Y 479.475,Z 1031.315,A -85,B 0,C 180,E1 12634.339,E2 12634.339} C_VEL
LIN {X 0,Y 485.01,Z 1011.337,A -85,B 0,C 180,E1 12633.282,E2 12633.282} C_VEL
LIN {X 0,Y 490.038,Z 991.156,A -85,B 0,C 180,E1 12632.367,E2 12632.367} C_VEL
LIN {X 0,Y 494.528,Z 970.741,A -85,B 0,C 180,E1 12631.579,E2 12631.579} C_VEL
LIN {X 0,Y 498.939,Z 947.49,A -85,B 0,C 180,E1 12630.837,E2 12630.837} C_VEL
LIN {X 0,Y 503.237,Z 918.762,A -85,B 0,C 180,E1 12630.13,E2 12630.13} C_VEL
LIN {X 0,Y 505.75,Z 895.255,A -85,B 0,C 180,E1 12629.69,E2 12629.69} C_VEL
LIN {X 0,Y 519.429,Z 688.219,A -85,B 0,C 180,E1 12626.455,E2 12626.455} C_VEL
LIN {X 0,Y 526.016,Z 590.955,A -85,B 0,C 180,E1 12624.934,E2 12624.934} C_VEL
LIN {X 0,Y 517.291,Z 577.81,A -85,B 0,C 180,E1 12622.293,E2 12622.293} C_VEL
LIN {X 0,Y 510.269,Z 567.827,A -85,B 0,C 180,E1 12619.876,E2 12619.876} C_VEL
LIN {X 0,Y 504.098,Z 559.185,A -85,B 0,C 180,E1 12617.428,E2 12617.428} C_VEL
LIN {X 0,Y 500.054,Z 553.815,A -85,B 0,C 180,E1 12615.601,E2 12615.601} C_VEL
LIN {X 0,Y 496.47,Z 548.928,A -85,B 0,C 180,E1 12613.748,E2 12613.748} C_VEL
LIN {X 0,Y 492.634,Z 543.807,A -85,B 0,C 180,E1 12611.412,E2 12611.412} C_VEL
LIN {X 0,Y 489.611,Z 540.167,A -85,B 0,C 180,E1 12609.166,E2 12609.166} C_VEL
LIN {X 0,Y 488.639,Z 538.271,A -85,B 0,C 180,E1 12608.235,E2 12608.235} C_VEL
LIN {X 0,Y 485.388,Z 534.855,A -85,B 0,C 180,E1 12604.253,E2 12604.253} C_VEL
LIN {X 0,Y 484.682,Z 532.294,A -85,B 0,C 180,E1 12602.01,E2 12602.01} C_VEL
LIN {X 0,Y 484.759,Z 532.553,A -85,B 0,C 180,E1 12597.754,E2 12597.754} C_VEL
LIN {X 0,Y 486.497,Z 536.583,A -85,B 0,C 180,E1 12594.102,E2 12594.102} C_VEL
LIN {X 0,Y 488.875,Z 538.608,A -85,B 0,C 180,E1 12591.65,E2 12591.65} C_VEL
LIN {X 0,Y 491.34,Z 542.644,A -85,B 0,C 180,E1 12589.565,E2 12589.565} C_VEL
LIN {X 0,Y 493.322,Z 544.649,A -85,B 0,C 180,E1 12588.247,E2 12588.247} C_VEL
LIN {X 0,Y 496.664,Z 549.131,A -85,B 0,C 180,E1 12586.257,E2 12586.257} C_VEL
LIN {X 0,Y 501.815,Z 556.178,A -85,B 0,C 180,E1 12583.683,E2 12583.683} C_VEL
LIN {X 0,Y 505.765,Z 561.628,A -85,B 0,C 180,E1 12581.977,E2 12581.977} C_VEL
LIN {X 0,Y 511.879,Z 570.011,A -85,B 0,C 180,E1 12579.653,E2 12579.653} C_VEL
LIN {X 0,Y 519.135,Z 581.528,A -85,B 0,C 180,E1 12577.193,E2 12577.193} C_VEL
LIN {X 0,Y 526.013,Z 593.053,A -85,B 0,C 180,E1 12575.109,E2 12575.109} C_VEL
LIN {X 0,Y 511.813,Z 805.893,A -85,B 0,C 180,E1 12571.795,E2 12571.795} C_VEL
LIN {X 0,Y 505.4,Z 902.624,A -85,B 0,C 180,E1 12570.272,E2 12570.272} C_VEL
LIN {X 0,Y 502.279,Z 930.36,A -85,B 0,C 180,E1 12569.739,E2 12569.739} C_VEL
LIN {X 0,Y 498.093,Z 956.264,A -85,B 0,C 180,E1 12569.076,E2 12569.076} C_VEL
LIN {X 0,Y 494.107,Z 976.968,A -85,B 0,C 180,E1 12568.413,E2 12568.413} C_VEL
LIN {X 0,Y 489.537,Z 997.522,A -85,B 0,C 180,E1 12567.627,E2 12567.627} C_VEL
LIN {X 0,Y 484.364,Z 1018.159,A -85,B 0,C 180,E1 12566.694,E2 12566.694} C_VEL
LIN {X 0,Y 477.48,Z 1042.823,A -85,B 0,C 180,E1 12565.374,E2 12565.374} C_VEL
LIN {X 0,Y 469.917,Z 1066.522,A -85,B 0,C 180,E1 12563.843,E2 12563.843} C_VEL
LIN {X 0,Y 463.228,Z 1085.98,A -85,B 0,C 180,E1 12562.38,E2 12562.38} C_VEL
LIN {X 0,Y 456.372,Z 1104.733,A -85,B 0,C 180,E1 12560.762,E2 12560.762} C_VEL
LIN {X 0,Y 447.939,Z 1126.595,A -85,B 0,C 180,E1 12558.583,E2 12558.583} C_VEL
LIN {X 0,Y 439.889,Z 1146.154,A -85,B 0,C 180,E1 12556.28,E2 12556.28} C_VEL
LIN {X 0,Y 433.13,Z 1162.217,A -85,B 0,C 180,E1 12554.114,E2 12554.114} C_VEL
LIN {X 0,Y 426.797,Z 1177.077,A -85,B 0,C 180,E1 12551.84,E2 12551.84} C_VEL
LIN {X 0,Y 419.393,Z 1194.575,A -85,B 0,C 180,E1 12548.774,E2 12548.774} C_VEL
LIN {X 0,Y 412.751,Z 1210.152,A -85,B 0,C 180,E1 12545.542,E2 12545.542} C_VEL
LIN {X 0,Y 407.995,Z 1221.76,A -85,B 0,C 180,E1 12542.787,E2 12542.787} C_VEL
LIN {X 0,Y 403.976,Z 1232.204,A -85,B 0,C 180,E1 12539.969,E2 12539.969} C_VEL
LIN {X 0,Y 400.064,Z 1243.201,A -85,B 0,C 180,E1 12536.57,E2 12536.57} C_VEL
LIN {X 0,Y 396.614,Z 1254.112,A -85,B 0,C 180,E1 12532.526,E2 12532.526} C_VEL
LIN {X 0,Y 394.618,Z 1261.527,A -85,B 0,C 180,E1 12529.227,E2 12529.227} C_VEL
LIN {X 0,Y 393.403,Z 1267.194,A -85,B 0,C 180,E1 12526.23,E2 12526.23} C_VEL
LIN {X 0,Y 392.574,Z 1272.074,A -85,B 0,C 180,E1 12523.097,E2 12523.097} C_VEL
LIN {X 0,Y 392.135,Z 1275.73,A -85,B 0,C 180,E1 12520.129,E2 12520.129} C_VEL
LIN {X 0,Y 391.981,Z 1278.441,A -85,B 0,C 180,E1 12517.176,E2 12517.176} C_VEL
LIN {X 0,Y 391.918,Z 1280.225,A -85,B 0,C 180,E1 12514.239,E2 12514.239} C_VEL
LIN {X 0,Y 391.902,Z 1281.068,A -85,B 0,C 180,E1 12511.458,E2 12511.458} C_VEL
LIN {X 0,Y 391.896,Z 1281.09,A -85,B 0,C 180,E1 12508.68,E2 12508.68} C_VEL
LIN {X 0,Y 391.918,Z 1280.289,A -85,B 0,C 180,E1 12505.9,E2 12505.9} C_VEL
LIN {X 0,Y 391.974,Z 1278.547,A -85,B 0,C 180,E1 12502.963,E2 12502.963} C_VEL
LIN {X 0,Y 392.116,Z 1275.879,A -85,B 0,C 180,E1 12500.011,E2 12500.011} C_VEL
LIN {X 0,Y 392.548,Z 1272.269,A -85,B 0,C 180,E1 12497.043,E2 12497.043} C_VEL
LIN {X 0,Y 393.354,Z 1267.434,A -85,B 0,C 180,E1 12493.911,E2 12493.911} C_VEL
LIN {X 0,Y 394.544,Z 1261.809,A -85,B 0,C 180,E1 12490.914,E2 12490.914} C_VEL
LIN {X 0,Y 396.511,Z 1254.439,A -85,B 0,C 180,E1 12487.615,E2 12487.615} C_VEL
LIN {X 0,Y 399.778,Z 1244.09,A -85,B 0,C 180,E1 12483.721,E2 12483.721} C_VEL
LIN {X 0,Y 403.823,Z 1232.612,A -85,B 0,C 180,E1 12480.15,E2 12480.15} C_VEL
LIN {X 0,Y 407.776,Z 1222.292,A -85,B 0,C 180,E1 12477.351,E2 12477.351} C_VEL
LIN {X 0,Y 412.491,Z 1210.734,A -85,B 0,C 180,E1 12474.593,E2 12474.593} C_VEL
LIN {X 0,Y 418.245,Z 1197.125,A -85,B 0,C 180,E1 12471.741,E2 12471.741} C_VEL
LIN {X 0,Y 426.182,Z 1178.492,A -85,B 0,C 180,E1 12468.395,E2 12468.395} C_VEL
LIN {X 0,Y 432.722,Z 1163.113,A -85,B 0,C 180,E1 12466.021,E2 12466.021} C_VEL
LIN {X 0,Y 439.319,Z 1147.432,A -85,B 0,C 180,E1 12463.89,E2 12463.89} C_VEL
LIN {X 0,Y 446.33,Z 1130.359,A -85,B 0,C 180,E1 12461.849,E2 12461.849} C_VEL
LIN {X 0,Y 455.122,Z 1107.982,A -85,B 0,C 180,E1 12459.542,E2 12459.542} C_VEL
LIN {X 0,Y 462.722,Z 1087.25,A -85,B 0,C 180,E1 12457.73,E2 12457.73} C_VEL
LIN {X 0,Y 469.12,Z 1068.737,A -85,B 0,C 180,E1 12456.322,E2 12456.322} C_VEL
LIN {X 0,Y 475.299,Z 1049.571,A -85,B 0,C 180,E1 12455.052,E2 12455.052} C_VEL
LIN {X 0,Y 481.832,Z 1027.35,A -85,B 0,C 180,E1 12453.774,E2 12453.774} C_VEL
LIN {X 0,Y 488.624,Z 1001.136,A -85,B 0,C 180,E1 12452.53,E2 12452.53} C_VEL
LIN {X 0,Y 493.501,Z 979.492,A -85,B 0,C 180,E1 12451.681,E2 12451.681} C_VEL
LIN {X 0,Y 497.596,Z 958.599,A -85,B 0,C 180,E1 12451,E2 12451} C_VEL
LIN {X 0,Y 501.172,Z 936.901,A -85,B 0,C 180,E1 12450.42,E2 12450.42} C_VEL
LIN {X 0,Y 504.721,Z 909.751,A -85,B 0,C 180,E1 12449.854,E2 12449.854} C_VEL
LIN {X 0,Y 507.874,Z 865.978,A -85,B 0,C 180,E1 12449.146,E2 12449.146} C_VEL
LIN {X 0,Y 522.136,Z 648.41,A -85,B 0,C 180,E1 12445.76,E2 12445.76} C_VEL
LIN {X 0,Y 525.856,Z 592.901,A -85,B 0,C 180,E1 12444.88,E2 12444.88} C_VEL
LIN {X 0,Y 518.536,Z 580.596,A -85,B 0,C 180,E1 12442.655,E2 12442.655} C_VEL
LIN {X 0,Y 511.153,Z 569.045,A -85,B 0,C 180,E1 12440.138,E2 12440.138} C_VEL
LIN {X 0,Y 503.925,Z 559.04,A -85,B 0,C 180,E1 12437.315,E2 12437.315} C_VEL
LIN {X 0,Y 499.992,Z 553.792,A -85,B 0,C 180,E1 12435.544,E2 12435.544} C_VEL
LIN {X 0,Y 496.28,Z 548.757,A -85,B 0,C 180,E1 12433.635,E2 12433.635} C_VEL
LIN {X 0,Y 492.52,Z 543.733,A -85,B 0,C 180,E1 12431.357,E2 12431.357} C_VEL
LIN {X 0,Y 489.474,Z 540,A -85,B 0,C 180,E1 12429.109,E2 12429.109} C_VEL
LIN {X 0,Y 488.546,Z 538.22,A -85,B 0,C 180,E1 12428.237,E2 12428.237} C_VEL
LIN {X 0,Y 485.288,Z 534.749,A -85,B 0,C 180,E1 12424.372,E2 12424.372} C_VEL
LIN {X 0,Y 484.565,Z 532.258,A -85,B 0,C 180,E1 12422.365,E2 12422.365} C_VEL
LIN {X 0,Y 484.653,Z 532.399,A -85,B 0,C 180,E1 12417.162,E2 12417.162} C_VEL
LIN {X 0,Y 486.046,Z 536.022,A -85,B 0,C 180,E1 12414.215,E2 12414.215} C_VEL
LIN {X 0,Y 488.774,Z 538.546,A -85,B 0,C 180,E1 12411.352,E2 12411.352} C_VEL
LIN {X 0,Y 491.371,Z 542.632,A -85,B 0,C 180,E1 12409.21,E2 12409.21} C_VEL
LIN {X 0,Y 493.199,Z 544.525,A -85,B 0,C 180,E1 12408.006,E2 12408.006} C_VEL
LIN {X 0,Y 496.563,Z 549.038,A -85,B 0,C 180,E1 12406.017,E2 12406.017} C_VEL
LIN {X 0,Y 501.749,Z 556.075,A -85,B 0,C 180,E1 12403.443,E2 12403.443} C_VEL
LIN {X 0,Y 505.851,Z 561.756,A -85,B 0,C 180,E1 12401.682,E2 12401.682} C_VEL
LIN {X 0,Y 511.708,Z 569.761,A -85,B 0,C 180,E1 12399.467,E2 12399.467} C_VEL
LIN {X 0,Y 520.154,Z 582.14,A -85,B 0,C 180,E1 12396.672,E2 12396.672} C_VEL
LIN {X 0,Y 525.934,Z 591.108,A -85,B 0,C 180,E1 12394.96,E2 12394.96} C_VEL
LIN {X 0,Y 511.335,Z 809.673,A -85,B 0,C 180,E1 12391.561,E2 12391.561} C_VEL
LIN {X 0,Y 505.488,Z 897.376,A -85,B 0,C 180,E1 12390.179,E2 12390.179} C_VEL
LIN {X 0,Y 502.352,Z 925.176,A -85,B 0,C 180,E1 12389.639,E2 12389.639} C_VEL
LIN {X 0,Y 498.306,Z 950.552,A -85,B 0,C 180,E1 12388.976,E2 12388.976} C_VEL
LIN {X 0,Y 494.212,Z 971.881,A -85,B 0,C 180,E1 12388.285,E2 12388.285} C_VEL
LIN {X 0,Y 489.701,Z 992.283,A -85,B 0,C 180,E1 12387.49,E2 12387.49} C_VEL
LIN {X 0,Y 484.072,Z 1014.693,A -85,B 0,C 180,E1 12386.458,E2 12386.458} C_VEL
LIN {X 0,Y 476.639,Z 1040.741,A -85,B 0,C 180,E1 12385.006,E2 12385.006} C_VEL
LIN {X 0,Y 470.259,Z 1060.676,A -85,B 0,C 180,E1 12383.694,E2 12383.694} C_VEL
LIN {X 0,Y 463.85,Z 1079.253,A -85,B 0,C 180,E1 12382.292,E2 12382.292} C_VEL
LIN {X 0,Y 457.219,Z 1097.337,A -85,B 0,C 180,E1 12380.731,E2 12380.731} C_VEL
LIN {X 0,Y 449.506,Z 1117.312,A -85,B 0,C 180,E1 12378.754,E2 12378.754} C_VEL
LIN {X 0,Y 440.811,Z 1138.456,A -85,B 0,C 180,E1 12376.292,E2 12376.292} C_VEL
LIN {X 0,Y 433.914,Z 1154.684,A -85,B 0,C 180,E1 12374.103,E2 12374.103} C_VEL
LIN {X 0,Y 427.464,Z 1169.619,A -85,B 0,C 180,E1 12371.812,E2 12371.812} C_VEL
LIN {X 0,Y 420.338,Z 1186.179,A -85,B 0,C 180,E1 12368.905,E2 12368.905} C_VEL
LIN {X 0,Y 413.51,Z 1201.942,A -85,B 0,C 180,E1 12365.647,E2 12365.647} C_VEL
LIN {X 0,Y 408.424,Z 1214.051,A -85,B 0,C 180,E1 12362.758,E2 12362.758} C_VEL
LIN {X 0,Y 404.381,Z 1224.292,A -85,B 0,C 180,E1 12359.968,E2 12359.968} C_VEL
LIN {X 0,Y 400.678,Z 1234.295,A -85,B 0,C 180,E1 12356.855,E2 12356.855} C_VEL
LIN {X 0,Y 397.061,Z 1245.263,A -85,B 0,C 180,E1 12352.821,E2 12352.821} C_VEL
LIN {X 0,Y 394.862,Z 1252.96,A -85,B 0,C 180,E1 12349.377,E2 12349.377} C_VEL
LIN {X 0,Y 393.524,Z 1258.835,A -85,B 0,C 180,E1 12346.234,E2 12346.234} C_VEL
LIN {X 0,Y 392.65,Z 1263.631,A -85,B 0,C 180,E1 12343.103,E2 12343.103} C_VEL
LIN {X 0,Y 392.179,Z 1267.223,A -85,B 0,C 180,E1 12340.136,E2 12340.136} C_VEL
LIN {X 0,Y 392.001,Z 1269.888,A -85,B 0,C 180,E1 12337.184,E2 12337.184} C_VEL
LIN {X 0,Y 391.924,Z 1271.647,A -85,B 0,C 180,E1 12334.247,E2 12334.247} C_VEL
LIN {X 0,Y 391.905,Z 1272.487,A -85,B 0,C 180,E1 12331.466,E2 12331.466} C_VEL
LIN {X 0,Y 391.892,Z 1272.525,A -85,B 0,C 180,E1 12328.688,E2 12328.688} C_VEL
LIN {X 0,Y 391.898,Z 1272.506,A -85,B 0,C 180,E1 12328.567,E2 12328.567} C_VEL
LIN {X 0,Y 390.943,Z 1272.355,A -85,B 0,C 180,E1 12327.44,E2 12327.44} C_VEL
LIN {X 0,Y 386.329,Z 1271.7,A -85,B 0,C 180,E1 12325.316,E2 12325.316} C_VEL
LIN {X 0,Y 384.112,Z 1270.934,A -85,B 0,C 180,E1 12323.855,E2 12323.855} C_VEL
LIN {X 0,Y 383.98,Z 1270.626,A -85,B 0,C 180,E1 12323.44,E2 12323.44} C_VEL
LIN {X 0,Y 384.142,Z 1267.892,A -85,B 0,C 180,E1 12320.113,E2 12320.113} C_VEL
LIN {X 0,Y 384.636,Z 1264.265,A -85,B 0,C 180,E1 12316.934,E2 12316.934} C_VEL
LIN {X 0,Y 385.564,Z 1259.344,A -85,B 0,C 180,E1 12313.586,E2 12313.586} C_VEL
LIN {X 0,Y 386.96,Z 1253.549,A -85,B 0,C 180,E1 12310.377,E2 12310.377} C_VEL
LIN {X 0,Y 389.116,Z 1246.284,A -85,B 0,C 180,E1 12307.015,E2 12307.015} C_VEL
LIN {X 0,Y 392.827,Z 1235.586,A -85,B 0,C 180,E1 12302.901,E2 12302.901} C_VEL
LIN {X 0,Y 397.024,Z 1224.702,A -85,B 0,C 180,E1 12299.427,E2 12299.427} C_VEL
LIN {X 0,Y 401.513,Z 1213.925,A -85,B 0,C 180,E1 12296.444,E2 12296.444} C_VEL
LIN {X 0,Y 406.968,Z 1201.552,A -85,B 0,C 180,E1 12293.458,E2 12293.458} C_VEL
LIN {X 0,Y 414.655,Z 1184.443,A -85,B 0,C 180,E1 12289.929,E2 12289.929} C_VEL
LIN {X 0,Y 421.449,Z 1169.38,A -85,B 0,C 180,E1 12287.279,E2 12287.279} C_VEL
LIN {X 0,Y 428.163,Z 1154.406,A -85,B 0,C 180,E1 12284.969,E2 12284.969} C_VEL
LIN {X 0,Y 435.705,Z 1137.3,A -85,B 0,C 180,E1 12282.658,E2 12282.658} C_VEL
LIN {X 0,Y 444.828,Z 1115.693,A -85,B 0,C 180,E1 12280.168,E2 12280.168} C_VEL
LIN {X 0,Y 452.324,Z 1096.877,A -85,B 0,C 180,E1 12278.312,E2 12278.312} C_VEL
LIN {X 0,Y 459.16,Z 1078.731,A -85,B 0,C 180,E1 12276.748,E2 12276.748} C_VEL
LIN {X 0,Y 466.345,Z 1058.376,A -85,B 0,C 180,E1 12275.223,E2 12275.223} C_VEL
LIN {X 0,Y 474.635,Z 1032.399,A -85,B 0,C 180,E1 12273.584,E2 12273.584} C_VEL
LIN {X 0,Y 480.694,Z 1011.08,A -85,B 0,C 180,E1 12272.457,E2 12272.457} C_VEL
LIN {X 0,Y 485.751,Z 991.236,A -85,B 0,C 180,E1 12271.56,E2 12271.56} C_VEL
LIN {X 0,Y 490.387,Z 970.65,A -85,B 0,C 180,E1 12270.77,E2 12270.77} C_VEL
LIN {X 0,Y 494.981,Z 946.915,A -85,B 0,C 180,E1 12270.018,E2 12270.018} C_VEL
LIN {X 0,Y 499.313,Z 918.346,A -85,B 0,C 180,E1 12269.323,E2 12269.323} C_VEL
LIN {X 0,Y 501.842,Z 895.105,A -85,B 0,C 180,E1 12268.89,E2 12268.89} C_VEL
LIN {X 0,Y 516.028,Z 686.447,A -85,B 0,C 180,E1 12265.628,E2 12265.628} C_VEL
LIN {X 0,Y 522.313,Z 595.889,A -85,B 0,C 180,E1 12264.206,E2 12264.206} C_VEL
LIN {X 0,Y 514.428,Z 583.906,A -85,B 0,C 180,E1 12261.727,E2 12261.727} C_VEL
LIN {X 0,Y 508.121,Z 574.79,A -85,B 0,C 180,E1 12259.484,E2 12259.484} C_VEL
LIN {X 0,Y 502.214,Z 566.426,A -85,B 0,C 180,E1 12257.078,E2 12257.078} C_VEL
LIN {X 0,Y 498.38,Z 561.234,A -85,B 0,C 180,E1 12255.297,E2 12255.297} C_VEL
LIN {X 0,Y 494.978,Z 556.516,A -85,B 0,C 180,E1 12253.493,E2 12253.493} C_VEL
LIN {X 0,Y 491.403,Z 551.617,A -85,B 0,C 180,E1 12251.265,E2 12251.265} C_VEL
LIN {X 0,Y 488.366,Z 547.856,A -85,B 0,C 180,E1 12248.952,E2 12248.952} C_VEL
LIN {X 0,Y 487.407,Z 546.09,A -85,B 0,C 180,E1 12248.019,E2 12248.019} C_VEL
LIN {X 0,Y 484.298,Z 542.592,A -85,B 0,C 180,E1 12244.025,E2 12244.025} C_VEL
LIN {X 0,Y 483.675,Z 540.228,A -85,B 0,C 180,E1 12241.896,E2 12241.896} C_VEL
LIN {X 0,Y 483.753,Z 540.435,A -85,B 0,C 180,E1 12237.868,E2 12237.868} C_VEL
LIN {X 0,Y 485.431,Z 544.464,A -85,B 0,C 180,E1 12234.207,E2 12234.207} C_VEL
LIN {X 0,Y 487.762,Z 546.573,A -85,B 0,C 180,E1 12231.75,E2 12231.75} C_VEL
LIN {X 0,Y 490.367,Z 550.701,A -85,B 0,C 180,E1 12229.544,E2 12229.544} C_VEL
LIN {X 0,Y 492.074,Z 552.494,A -85,B 0,C 180,E1 12228.395,E2 12228.395} C_VEL
LIN {X 0,Y 496.184,Z 558.216,A -85,B 0,C 180,E1 12225.946,E2 12225.946} C_VEL
LIN {X 0,Y 500.343,Z 563.905,A -85,B 0,C 180,E1 12223.872,E2 12223.872} C_VEL
LIN {X 0,Y 504.112,Z 569.182,A -85,B 0,C 180,E1 12222.214,E2 12222.214} C_VEL
LIN {X 0,Y 509.99,Z 577.384,A -85,B 0,C 180,E1 12219.934,E2 12219.934} C_VEL
LIN {X 0,Y 517.135,Z 588.955,A -85,B 0,C 180,E1 12217.46,E2 12217.46} C_VEL
LIN {X 0,Y 522.348,Z 597.865,A -85,B 0,C 180,E1 12215.83,E2 12215.83} C_VEL
LIN {X 0,Y 507.298,Z 817.335,A -85,B 0,C 180,E1 12212.414,E2 12212.414} C_VEL
LIN {X 0,Y 501.439,Z 902.852,A -85,B 0,C 180,E1 12211.064,E2 12211.064} C_VEL
LIN {X 0,Y 498.171,Z 930.936,A -85,B 0,C 180,E1 12210.523,E2 12210.523} C_VEL
LIN {X 0,Y 493.95,Z 956.422,A -85,B 0,C 180,E1 12209.872,E2 12209.872} C_VEL
LIN {X 0,Y 489.918,Z 976.888,A -85,B 0,C 180,E1 12209.219,E2 12209.219} C_VEL
LIN {X 0,Y 485.27,Z 997.318,A -85,B 0,C 180,E1 12208.442,E2 12208.442} C_VEL
LIN {X 0,Y 480.001,Z 1017.848,A -85,B 0,C 180,E1 12207.517,E2 12207.517} C_VEL
LIN {X 0,Y 473.063,Z 1042.104,A -85,B 0,C 180,E1 12206.228,E2 12206.228} C_VEL
LIN {X 0,Y 465.182,Z 1066.231,A -85,B 0,C 180,E1 12204.675,E2 12204.675} C_VEL
LIN {X 0,Y 458.51,Z 1085.157,A -85,B 0,C 180,E1 12203.256,E2 12203.256} C_VEL
LIN {X 0,Y 451.692,Z 1103.323,A -85,B 0,C 180,E1 12201.697,E2 12201.697} C_VEL
LIN {X 0,Y 444.413,Z 1121.692,A -85,B 0,C 180,E1 12199.895,E2 12199.895} C_VEL
LIN {X 0,Y 434.909,Z 1144.363,A -85,B 0,C 180,E1 12197.294,E2 12197.294} C_VEL
LIN {X 0,Y 427.536,Z 1161.267,A -85,B 0,C 180,E1 12195.021,E2 12195.021} C_VEL
LIN {X 0,Y 421.039,Z 1175.945,A -85,B 0,C 180,E1 12192.773,E2 12192.773} C_VEL
LIN {X 0,Y 414.597,Z 1190.415,A -85,B 0,C 180,E1 12190.259,E2 12190.259} C_VEL
LIN {X 0,Y 407.066,Z 1207.505,A -85,B 0,C 180,E1 12186.816,E2 12186.816} C_VEL
LIN {X 0,Y 401.381,Z 1220.679,A -85,B 0,C 180,E1 12183.691,E2 12183.691} C_VEL
LIN {X 0,Y 396.943,Z 1231.522,A -85,B 0,C 180,E1 12180.747,E2 12180.747} C_VEL
LIN {X 0,Y 393.238,Z 1241.26,A -85,B 0,C 180,E1 12177.724,E2 12177.724} C_VEL
LIN {X 0,Y 389.633,Z 1251.85,A -85,B 0,C 180,E1 12173.914,E2 12173.914} C_VEL
LIN {X 0,Y 386.987,Z 1260.825,A -85,B 0,C 180,E1 12169.936,E2 12169.936} C_VEL
LIN {X 0,Y 385.566,Z 1266.848,A -85,B 0,C 180,E1 12166.724,E2 12166.724} C_VEL
LIN {X 0,Y 384.667,Z 1271.777,A -85,B 0,C 180,E1 12163.524,E2 12163.524} C_VEL
LIN {X 0,Y 384.187,Z 1275.48,A -85,B 0,C 180,E1 12160.492,E2 12160.492} C_VEL
LIN {X 0,Y 383.979,Z 1278.238,A -85,B 0,C 180,E1 12157.477,E2 12157.477} C_VEL
LIN {X 0,Y 383.921,Z 1280,A -85,B 0,C 180,E1 12154.626,E2 12154.626} C_VEL
LIN {X 0,Y 383.909,Z 1280.935,A -85,B 0,C 180,E1 12151.787,E2 12151.787} C_VEL
LIN {X 0,Y 383.889,Z 1281.025,A -85,B 0,C 180,E1 12148.802,E2 12148.802} C_VEL
LIN {X 0,Y 383.919,Z 1280.201,A -85,B 0,C 180,E1 12145.814,E2 12145.814} C_VEL
LIN {X 0,Y 383.981,Z 1278.453,A -85,B 0,C 180,E1 12142.808,E2 12142.808} C_VEL
LIN {X 0,Y 384.157,Z 1275.677,A -85,B 0,C 180,E1 12139.695,E2 12139.695} C_VEL
LIN {X 0,Y 384.635,Z 1271.97,A -85,B 0,C 180,E1 12136.619,E2 12136.619} C_VEL
LIN {X 0,Y 385.518,Z 1267.086,A -85,B 0,C 180,E1 12133.42,E2 12133.42} C_VEL
LIN {X 0,Y 386.94,Z 1260.999,A -85,B 0,C 180,E1 12130.155,E2 12130.155} C_VEL
LIN {X 0,Y 389.52,Z 1252.206,A -85,B 0,C 180,E1 12126.23,E2 12126.23} C_VEL
LIN {X 0,Y 393.085,Z 1241.686,A -85,B 0,C 180,E1 12122.419,E2 12122.419} C_VEL
LIN {X 0,Y 396.751,Z 1232,A -85,B 0,C 180,E1 12119.394,E2 12119.394} C_VEL
LIN {X 0,Y 400.964,Z 1221.621,A -85,B 0,C 180,E1 12116.554,E2 12116.554} C_VEL
LIN {X 0,Y 406.268,Z 1209.268,A -85,B 0,C 180,E1 12113.591,E2 12113.591} C_VEL
LIN {X 0,Y 413.604,Z 1192.656,A -85,B 0,C 180,E1 12110.158,E2 12110.158} C_VEL
LIN {X 0,Y 420.674,Z 1176.698,A -85,B 0,C 180,E1 12107.356,E2 12107.356} C_VEL
LIN {X 0,Y 427.344,Z 1161.624,A -85,B 0,C 180,E1 12105.037,E2 12105.037} C_VEL
LIN {X 0,Y 434.394,Z 1145.432,A -85,B 0,C 180,E1 12102.848,E2 12102.848} C_VEL
LIN {X 0,Y 443.461,Z 1123.974,A -85,B 0,C 180,E1 12100.348,E2 12100.348} C_VEL
LIN {X 0,Y 451.167,Z 1104.537,A -85,B 0,C 180,E1 12098.421,E2 12098.421} C_VEL
LIN {X 0,Y 457.956,Z 1086.494,A -85,B 0,C 180,E1 12096.859,E2 12096.859} C_VEL
LIN {X 0,Y 464.566,Z 1067.829,A -85,B 0,C 180,E1 12095.445,E2 12095.445} C_VEL
LIN {X 0,Y 471.46,Z 1046.91,A -85,B 0,C 180,E1 12094.074,E2 12094.074} C_VEL
LIN {X 0,Y 479.117,Z 1020.913,A -85,B 0,C 180,E1 12092.637,E2 12092.637} C_VEL
LIN {X 0,Y 484.918,Z 998.465,A -85,B 0,C 180,E1 12091.612,E2 12091.612} C_VEL
LIN {X 0,Y 489.615,Z 977.922,A -85,B 0,C 180,E1 12090.823,E2 12090.823} C_VEL
LIN {X 0,Y 493.797,Z 956.804,A -85,B 0,C 180,E1 12090.146,E2 12090.146} C_VEL
LIN {X 0,Y 497.833,Z 932.495,A -85,B 0,C 180,E1 12089.519,E2 12089.519} C_VEL
LIN {X 0,Y 501.288,Z 903.576,A -85,B 0,C 180,E1 12088.954,E2 12088.954} C_VEL
LIN {X 0,Y 506.193,Z 832.617,A -85,B 0,C 180,E1 12087.83,E2 12087.83} C_VEL
LIN {X 0,Y 520.888,Z 616.873,A -85,B 0,C 180,E1 12084.47,E2 12084.47} C_VEL
LIN {X 0,Y 522.206,Z 597.58,A -85,B 0,C 180,E1 12084.16,E2 12084.16} C_VEL
LIN {X 0,Y 515.014,Z 585.64,A -85,B 0,C 180,E1 12081.886,E2 12081.886} C_VEL
LIN {X 0,Y 509.124,Z 576.219,A -85,B 0,C 180,E1 12079.803,E2 12079.803} C_VEL
LIN {X 0,Y 502.168,Z 566.431,A -85,B 0,C 180,E1 12077.02,E2 12077.02} C_VEL
LIN {X 0,Y 498.313,Z 561.209,A -85,B 0,C 180,E1 12075.24,E2 12075.24} C_VEL
LIN {X 0,Y 494.786,Z 556.341,A -85,B 0,C 180,E1 12073.379,E2 12073.379} C_VEL
LIN {X 0,Y 491.374,Z 551.612,A -85,B 0,C 180,E1 12071.265,E2 12071.265} C_VEL
LIN {X 0,Y 488.289,Z 547.81,A -85,B 0,C 180,E1 12068.953,E2 12068.953} C_VEL
LIN {X 0,Y 487.31,Z 546.034,A -85,B 0,C 180,E1 12068.02,E2 12068.02} C_VEL
LIN {X 0,Y 484.189,Z 542.48,A -85,B 0,C 180,E1 12064.145,E2 12064.145} C_VEL
LIN {X 0,Y 483.55,Z 540.191,A -85,B 0,C 180,E1 12062.252,E2 12062.252} C_VEL
LIN {X 0,Y 483.638,Z 540.289,A -85,B 0,C 180,E1 12057.274,E2 12057.274} C_VEL
LIN {X 0,Y 485.069,Z 544.014,A -85,B 0,C 180,E1 12054.203,E2 12054.203} C_VEL
LIN {X 0,Y 487.659,Z 546.511,A -85,B 0,C 180,E1 12051.451,E2 12051.451} C_VEL
LIN {X 0,Y 490.235,Z 550.519,A -85,B 0,C 180,E1 12049.304,E2 12049.304} C_VEL
LIN {X 0,Y 491.948,Z 552.379,A -85,B 0,C 180,E1 12048.154,E2 12048.154} C_VEL
LIN {X 0,Y 495.382,Z 556.937,A -85,B 0,C 180,E1 12046.102,E2 12046.102} C_VEL
LIN {X 0,Y 500.275,Z 563.805,A -85,B 0,C 180,E1 12043.631,E2 12043.631} C_VEL
LIN {X 0,Y 504.193,Z 569.311,A -85,B 0,C 180,E1 12041.919,E2 12041.919} C_VEL
LIN {X 0,Y 509.819,Z 577.137,A -85,B 0,C 180,E1 12039.747,E2 12039.747} C_VEL
LIN {X 0,Y 518.567,Z 590.106,A -85,B 0,C 180,E1 12036.807,E2 12036.807} C_VEL
LIN {X 0,Y 522.237,Z 596.123,A -85,B 0,C 180,E1 12035.682,E2 12035.682} C_VEL
LIN {X 0,Y 507.34,Z 813.145,A -85,B 0,C 180,E1 12032.305,E2 12032.305} C_VEL
LIN {X 0,Y 501.539,Z 897.594,A -85,B 0,C 180,E1 12030.972,E2 12030.972} C_VEL
LIN {X 0,Y 498.29,Z 925.613,A -85,B 0,C 180,E1 12030.428,E2 12030.428} C_VEL
LIN {X 0,Y 494.185,Z 950.761,A -85,B 0,C 180,E1 12029.773,E2 12029.773} C_VEL
LIN {X 0,Y 490.052,Z 971.832,A -85,B 0,C 180,E1 12029.092,E2 12029.092} C_VEL
LIN {X 0,Y 485.397,Z 992.381,A -85,B 0,C 180,E1 12028.296,E2 12028.296} C_VEL
LIN {X 0,Y 479.633,Z 1014.79,A -85,B 0,C 180,E1 12027.266,E2 12027.266} C_VEL
LIN {X 0,Y 472.035,Z 1040.747,A -85,B 0,C 180,E1 12025.823,E2 12025.823} C_VEL
LIN {X 0,Y 465.452,Z 1060.771,A -85,B 0,C 180,E1 12024.508,E2 12024.508} C_VEL
LIN {X 0,Y 458.869,Z 1079.348,A -85,B 0,C 180,E1 12023.104,E2 12023.104} C_VEL
LIN {X 0,Y 452.048,Z 1097.432,A -85,B 0,C 180,E1 12021.54,E2 12021.54} C_VEL
LIN {X 0,Y 444.575,Z 1116.196,A -85,B 0,C 180,E1 12019.682,E2 12019.682} C_VEL
LIN {X 0,Y 435.251,Z 1138.219,A -85,B 0,C 180,E1 12017.127,E2 12017.127} C_VEL
LIN {X 0,Y 427.961,Z 1154.779,A -85,B 0,C 180,E1 12014.88,E2 12014.88} C_VEL
LIN {X 0,Y 421.268,Z 1169.714,A -85,B 0,C 180,E1 12012.57,E2 12012.57} C_VEL
LIN {X 0,Y 414.17,Z 1185.508,A -85,B 0,C 180,E1 12009.777,E2 12009.777} C_VEL
LIN {X 0,Y 406.732,Z 1202.036,A -85,B 0,C 180,E1 12006.335,E2 12006.335} C_VEL
LIN {X 0,Y 401.41,Z 1214.145,A -85,B 0,C 180,E1 12003.404,E2 12003.404} C_VEL
LIN {X 0,Y 397.13,Z 1224.424,A -85,B 0,C 180,E1 12000.561,E2 12000.561} C_VEL
LIN {X 0,Y 393.249,Z 1234.388,A -85,B 0,C 180,E1 11997.404,E2 11997.404} C_VEL
LIN {X 0,Y 389.417,Z 1245.355,A -85,B 0,C 180,E1 11993.296,E2 11993.296} C_VEL
LIN {X 0,Y 387.091,Z 1253.051,A -85,B 0,C 180,E1 11989.782,E2 11989.782} C_VEL
LIN {X 0,Y 385.653,Z 1258.926,A -85,B 0,C 180,E1 11986.574,E2 11986.574} C_VEL
LIN {X 0,Y 384.72,Z 1263.721,A -85,B 0,C 180,E1 11983.378,E2 11983.378} C_VEL
LIN {X 0,Y 384.214,Z 1267.312,A -85,B 0,C 180,E1 11980.348,E2 11980.348} C_VEL
LIN {X 0,Y 384.005,Z 1269.977,A -85,B 0,C 180,E1 11977.334,E2 11977.334} C_VEL
LIN {X 0,Y 383.925,Z 1271.735,A -85,B 0,C 180,E1 11974.336,E2 11974.336} C_VEL
LIN {X 0,Y 383.906,Z 1272.575,A -85,B 0,C 180,E1 11971.497,E2 11971.497} C_VEL
LIN {X 0,Y 383.894,Z 1272.612,A -85,B 0,C 180,E1 11968.661,E2 11968.661} C_VEL
LIN {X 0,Y 383.927,Z 1271.781,A -85,B 0,C 180,E1 11965.673,E2 11965.673} C_VEL
LIN {X 0,Y 383.98,Z 1270.626,A -85,B 0,C 180,E1 11963.44,E2 11963.44} C_VEL
LIN {X 0,Y 383.028,Z 1269.834,A -85,B 0,C 180,E1 11962.298,E2 11962.298} C_VEL
LIN {X 0,Y 376.824,Z 1267.134,A -85,B 0,C 180,E1 11959.073,E2 11959.073} C_VEL
LIN {X 0,Y 376.41,Z 1266.277,A -85,B 0,C 180,E1 11958.235,E2 11958.235} C_VEL
LIN {X 0,Y 377.41,Z 1260.691,A -85,B 0,C 180,E1 11954.012,E2 11954.012} C_VEL
LIN {X 0,Y 378.934,Z 1254.538,A -85,B 0,C 180,E1 11950.426,E2 11950.426} C_VEL
LIN {X 0,Y 381.068,Z 1247.597,A -85,B 0,C 180,E1 11947.073,E2 11947.073} C_VEL
LIN {X 0,Y 383.943,Z 1239.436,A -85,B 0,C 180,E1 11943.728,E2 11943.728} C_VEL
LIN {X 0,Y 388.599,Z 1227.857,A -85,B 0,C 180,E1 11939.72,E2 11939.72} C_VEL
LIN {X 0,Y 393.787,Z 1215.722,A -85,B 0,C 180,E1 11936.222,E2 11936.222} C_VEL
LIN {X 0,Y 398.957,Z 1204.405,A -85,B 0,C 180,E1 11933.388,E2 11933.388} C_VEL
LIN {X 0,Y 404.543,Z 1192.45,A -85,B 0,C 180,E1 11930.755,E2 11930.755} C_VEL
LIN {X 0,Y 411.171,Z 1178.403,A -85,B 0,C 180,E1 11928.037,E2 11928.037} C_VEL
LIN {X 0,Y 420.203,Z 1159.101,A -85,B 0,C 180,E1 11924.846,E2 11924.846} C_VEL
LIN {X 0,Y 427.861,Z 1142.319,A -85,B 0,C 180,E1 11922.484,E2 11922.484} C_VEL
LIN {X 0,Y 435.084,Z 1126.062,A -85,B 0,C 180,E1 11920.484,E2 11920.484} C_VEL
LIN {X 0,Y 442.682,Z 1108.246,A -85,B 0,C 180,E1 11918.565,E2 11918.565} C_VEL
LIN {X 0,Y 452.101,Z 1084.675,A -85,B 0,C 180,E1 11916.396,E2 11916.396} C_VEL
LIN {X 0,Y 459.641,Z 1064.206,A -85,B 0,C 180,E1 11914.805,E2 11914.805} C_VEL
LIN {X 0,Y 466.027,Z 1045.519,A -85,B 0,C 180,E1 11913.545,E2 11913.545} C_VEL
LIN {X 0,Y 472.283,Z 1025.464,A -85,B 0,C 180,E1 11912.367,E2 11912.367} C_VEL
LIN {X 0,Y 479.362,Z 1000.412,A -85,B 0,C 180,E1 11911.125,E2 11911.125} C_VEL
LIN {X 0,Y 485.375,Z 975.013,A -85,B 0,C 180,E1 11910.104,E2 11910.104} C_VEL
LIN {X 0,Y 489.74,Z 953.706,A -85,B 0,C 180,E1 11909.404,E2 11909.404} C_VEL
LIN {X 0,Y 493.364,Z 932.585,A -85,B 0,C 180,E1 11908.831,E2 11908.831} C_VEL
LIN {X 0,Y 496.621,Z 909.008,A -85,B 0,C 180,E1 11908.327,E2 11908.327} C_VEL
LIN {X 0,Y 499.703,Z 873.084,A -85,B 0,C 180,E1 11907.724,E2 11907.724} C_VEL
LIN {X 0,Y 514.974,Z 653.357,A -85,B 0,C 180,E1 11904.303,E2 11904.303} C_VEL
LIN {X 0,Y 518.752,Z 600.909,A -85,B 0,C 180,E1 11903.485,E2 11903.485} C_VEL
LIN {X 0,Y 510.514,Z 588.262,A -85,B 0,C 180,E1 11900.763,E2 11900.763} C_VEL
LIN {X 0,Y 503.948,Z 578.768,A -85,B 0,C 180,E1 11898.27,E2 11898.27} C_VEL
LIN {X 0,Y 499.492,Z 572.514,A -85,B 0,C 180,E1 11896.335,E2 11896.335} C_VEL
LIN {X 0,Y 496.833,Z 568.787,A -85,B 0,C 180,E1 11895.047,E2 11895.047} C_VEL
LIN {X 0,Y 493.497,Z 564.1,A -85,B 0,C 180,E1 11893.236,E2 11893.236} C_VEL
LIN {X 0,Y 490.086,Z 559.353,A -85,B 0,C 180,E1 11891.057,E2 11891.057} C_VEL
LIN {X 0,Y 487.067,Z 555.423,A -85,B 0,C 180,E1 11888.678,E2 11888.678} C_VEL
LIN {X 0,Y 486.31,Z 553.979,A -85,B 0,C 180,E1 11887.918,E2 11887.918} C_VEL
LIN {X 0,Y 483.265,Z 550.471,A -85,B 0,C 180,E1 11883.915,E2 11883.915} C_VEL
LIN {X 0,Y 482.67,Z 548.163,A -85,B 0,C 180,E1 11881.781,E2 11881.781} C_VEL
LIN {X 0,Y 482.748,Z 548.317,A -85,B 0,C 180,E1 11877.982,E2 11877.982} C_VEL
LIN {X 0,Y 484.457,Z 552.441,A -85,B 0,C 180,E1 11874.196,E2 11874.196} C_VEL
LIN {X 0,Y 486.596,Z 554.397,A -85,B 0,C 180,E1 11871.908,E2 11871.908} C_VEL
LIN {X 0,Y 489.234,Z 558.586,A -85,B 0,C 180,E1 11869.639,E2 11869.639} C_VEL
LIN {X 0,Y 490.829,Z 560.337,A -85,B 0,C 180,E1 11868.544,E2 11868.544} C_VEL
LIN {X 0,Y 494.681,Z 565.759,A -85,B 0,C 180,E1 11866.201,E2 11866.201} C_VEL
LIN {X 0,Y 498.878,Z 571.628,A -85,B 0,C 180,E1 11864.063,E2 11864.063} C_VEL
LIN {X 0,Y 502.726,Z 577.115,A -85,B 0,C 180,E1 11862.343,E2 11862.343} C_VEL
LIN {X 0,Y 508.257,Z 584.989,A -85,B 0,C 180,E1 11860.162,E2 11860.162} C_VEL
LIN {X 0,Y 515.306,Z 596.647,A -85,B 0,C 180,E1 11857.677,E2 11857.677} C_VEL
LIN {X 0,Y 518.743,Z 602.777,A -85,B 0,C 180,E1 11856.563,E2 11856.563} C_VEL
LIN {X 0,Y 503.335,Z 821.536,A -85,B 0,C 180,E1 11853.158,E2 11853.158} C_VEL
LIN {X 0,Y 497.591,Z 902.896,A -85,B 0,C 180,E1 11851.872,E2 11851.872} C_VEL
LIN {X 0,Y 494.219,Z 931.121,A -85,B 0,C 180,E1 11851.329,E2 11851.329} C_VEL
LIN {X 0,Y 489.928,Z 956.462,A -85,B 0,C 180,E1 11850.684,E2 11850.684} C_VEL
LIN {X 0,Y 485.667,Z 977.55,A -85,B 0,C 180,E1 11850.013,E2 11850.013} C_VEL
LIN {X 0,Y 480.91,Z 997.902,A -85,B 0,C 180,E1 11849.238,E2 11849.238} C_VEL
LIN {X 0,Y 475.217,Z 1019.46,A -85,B 0,C 180,E1 11848.263,E2 11848.263} C_VEL
LIN {X 0,Y 467.464,Z 1045.369,A -85,B 0,C 180,E1 11846.856,E2 11846.856} C_VEL
LIN {X 0,Y 460.115,Z 1067.166,A -85,B 0,C 180,E1 11845.438,E2 11845.438} C_VEL
LIN {X 0,Y 453.346,Z 1085.808,A -85,B 0,C 180,E1 11844.032,E2 11844.032} C_VEL
LIN {X 0,Y 446.267,Z 1104.099,A -85,B 0,C 180,E1 11842.451,E2 11842.451} C_VEL
LIN {X 0,Y 437.954,Z 1124.424,A -85,B 0,C 180,E1 11840.433,E2 11840.433} C_VEL
LIN {X 0,Y 428.902,Z 1145.126,A -85,B 0,C 180,E1 11838.004,E2 11838.004} C_VEL
LIN {X 0,Y 421.517,Z 1161.487,A -85,B 0,C 180,E1 11835.781,E2 11835.781} C_VEL
LIN {X 0,Y 414.523,Z 1176.705,A -85,B 0,C 180,E1 11833.421,E2 11833.421} C_VEL
LIN {X 0,Y 406.823,Z 1193.424,A -85,B 0,C 180,E1 11830.448,E2 11830.448} C_VEL
LIN {X 0,Y 399.456,Z 1209.332,A -85,B 0,C 180,E1 11827.096,E2 11827.096} C_VEL
LIN {X 0,Y 394.129,Z 1221.226,A -85,B 0,C 180,E1 11824.203,E2 11824.203} C_VEL
LIN {X 0,Y 389.53,Z 1231.95,A -85,B 0,C 180,E1 11821.226,E2 11821.226} C_VEL
LIN {X 0,Y 385.325,Z 1242.557,A -85,B 0,C 180,E1 11817.839,E2 11817.839} C_VEL
LIN {X 0,Y 381.282,Z 1253.932,A -85,B 0,C 180,E1 11813.485,E2 11813.485} C_VEL
LIN {X 0,Y 379.041,Z 1261.347,A -85,B 0,C 180,E1 11810.05,E2 11810.05} C_VEL
LIN {X 0,Y 377.582,Z 1267.273,A -85,B 0,C 180,E1 11806.772,E2 11806.772} C_VEL
LIN {X 0,Y 376.627,Z 1272.314,A -85,B 0,C 180,E1 11803.349,E2 11803.349} C_VEL
LIN {X 0,Y 376.097,Z 1276.36,A -85,B 0,C 180,E1 11799.792,E2 11799.792} C_VEL
LIN {X 0,Y 375.94,Z 1279.429,A -85,B 0,C 180,E1 11795.796,E2 11795.796} C_VEL
LIN {X 0,Y 375.911,Z 1280.801,A -85,B 0,C 180,E1 11792.13,E2 11792.13} C_VEL
LIN {X 0,Y 375.875,Z 1280.983,A -85,B 0,C 180,E1 11789.081,E2 11789.081} C_VEL
LIN {X 0,Y 375.919,Z 1280.182,A -85,B 0,C 180,E1 11785.877,E2 11785.877} C_VEL
LIN {X 0,Y 375.982,Z 1278.423,A -85,B 0,C 180,E1 11782.732,E2 11782.732} C_VEL
LIN {X 0,Y 376.175,Z 1275.69,A -85,B 0,C 180,E1 11779.571,E2 11779.571} C_VEL
LIN {X 0,Y 376.663,Z 1272.089,A -85,B 0,C 180,E1 11776.487,E2 11776.487} C_VEL
LIN {X 0,Y 377.583,Z 1267.253,A -85,B 0,C 180,E1 11773.219,E2 11773.219} C_VEL
LIN {X 0,Y 379.045,Z 1261.321,A -85,B 0,C 180,E1 11769.941,E2 11769.941} C_VEL
LIN {X 0,Y 381.405,Z 1253.542,A -85,B 0,C 180,E1 11766.349,E2 11766.349} C_VEL
LIN {X 0,Y 385.501,Z 1242.056,A -85,B 0,C 180,E1 11761.997,E2 11761.997} C_VEL
LIN {X 0,Y 389.541,Z 1231.907,A -85,B 0,C 180,E1 11758.765,E2 11758.765} C_VEL
LIN {X 0,Y 394.126,Z 1221.21,A -85,B 0,C 180,E1 11755.798,E2 11755.798} C_VEL
LIN {X 0,Y 399.762,Z 1208.628,A -85,B 0,C 180,E1 11752.747,E2 11752.747} C_VEL
LIN {X 0,Y 407.876,Z 1191.012,A -85,B 0,C 180,E1 11749.112,E2 11749.112} C_VEL
LIN {X 0,Y 414.608,Z 1176.451,A -85,B 0,C 180,E1 11746.545,E2 11746.545} C_VEL
LIN {X 0,Y 421.493,Z 1161.459,A -85,B 0,C 180,E1 11744.223,E2 11744.223} C_VEL
LIN {X 0,Y 428.872,Z 1145.096,A -85,B 0,C 180,E1 11742,E2 11742} C_VEL
LIN {X 0,Y 438.289,Z 1123.472,A -85,B 0,C 180,E1 11739.477,E2 11739.477} C_VEL
LIN {X 0,Y 446.222,Z 1104.058,A -85,B 0,C 180,E1 11737.553,E2 11737.553} C_VEL
LIN {X 0,Y 453.085,Z 1086.323,A -85,B 0,C 180,E1 11736.018,E2 11736.018} C_VEL
LIN {X 0,Y 460.131,Z 1066.92,A -85,B 0,C 180,E1 11734.552,E2 11734.552} C_VEL
LIN {X 0,Y 468.085,Z 1043.295,A -85,B 0,C 180,E1 11733.023,E2 11733.023} C_VEL
LIN {X 0,Y 475.354,Z 1018.664,A -85,B 0,C 180,E1 11731.705,E2 11731.705} C_VEL
LIN {X 0,Y 480.837,Z 997.862,A -85,B 0,C 180,E1 11730.767,E2 11730.767} C_VEL
LIN {X 0,Y 485.521,Z 977.817,A -85,B 0,C 180,E1 11730.003,E2 11730.003} C_VEL
LIN {X 0,Y 489.786,Z 956.751,A -85,B 0,C 180,E1 11729.331,E2 11729.331} C_VEL
LIN {X 0,Y 493.897,Z 932.525,A -85,B 0,C 180,E1 11728.71,E2 11728.71} C_VEL
LIN {X 0,Y 497.446,Z 903.468,A -85,B 0,C 180,E1 11728.144,E2 11728.144} C_VEL
LIN {X 0,Y 502.514,Z 832.123,A -85,B 0,C 180,E1 11727.013,E2 11727.013} C_VEL
LIN {X 0,Y 517.627,Z 616.476,A -85,B 0,C 180,E1 11723.655,E2 11723.655} C_VEL
LIN {X 0,Y 518.627,Z 602.395,A -85,B 0,C 180,E1 11723.431,E2 11723.431} C_VEL
LIN {X 0,Y 510.847,Z 589.284,A -85,B 0,C 180,E1 11720.839,E2 11720.839} C_VEL
LIN {X 0,Y 506.537,Z 582.614,A -85,B 0,C 180,E1 11719.248,E2 11719.248} C_VEL
LIN {X 0,Y 500.425,Z 573.819,A -85,B 0,C 180,E1 11716.722,E2 11716.722} C_VEL
LIN {X 0,Y 496.761,Z 568.761,A -85,B 0,C 180,E1 11714.99,E2 11714.99} C_VEL
LIN {X 0,Y 493.404,Z 564.033,A -85,B 0,C 180,E1 11713.178,E2 11713.178} C_VEL
LIN {X 0,Y 490.052,Z 559.346,A -85,B 0,C 180,E1 11711.058,E2 11711.058} C_VEL
LIN {X 0,Y 486.983,Z 555.376,A -85,B 0,C 180,E1 11708.68,E2 11708.68} C_VEL
LIN {X 0,Y 486.211,Z 553.921,A -85,B 0,C 180,E1 11707.92,E2 11707.92} C_VEL
LIN {X 0,Y 483.151,Z 550.36,A -85,B 0,C 180,E1 11704.035,E2 11704.035} C_VEL
LIN {X 0,Y 482.536,Z 548.124,A -85,B 0,C 180,E1 11702.138,E2 11702.138} C_VEL
LIN {X 0,Y 482.649,Z 548.356,A -85,B 0,C 180,E1 11697.269,E2 11697.269} C_VEL
LIN {X 0,Y 484.179,Z 552.126,A -85,B 0,C 180,E1 11694.073,E2 11694.073} C_VEL
LIN {X 0,Y 486.491,Z 554.335,A -85,B 0,C 180,E1 11691.609,E2 11691.609} C_VEL
LIN {X 0,Y 489.1,Z 558.405,A -85,B 0,C 180,E1 11689.398,E2 11689.398} C_VEL
LIN {X 0,Y 490.701,Z 560.228,A -85,B 0,C 180,E1 11688.302,E2 11688.302} C_VEL
LIN {X 0,Y 494.689,Z 565.779,A -85,B 0,C 180,E1 11685.903,E2 11685.903} C_VEL
LIN {X 0,Y 498.69,Z 571.352,A -85,B 0,C 180,E1 11683.877,E2 11683.877} C_VEL
LIN {X 0,Y 502.937,Z 577.429,A -85,B 0,C 180,E1 11681.992,E2 11681.992} C_VEL
LIN {X 0,Y 508.374,Z 585.205,A -85,B 0,C 180,E1 11679.867,E2 11679.867} C_VEL
LIN {X 0,Y 516.559,Z 597.528,A -85,B 0,C 180,E1 11677.073,E2 11677.073} C_VEL
LIN {X 0,Y 518.629,Z 601.076,A -85,B 0,C 180,E1 11676.415,E2 11676.415} C_VEL
LIN {X 0,Y 503.428,Z 816.693,A -85,B 0,C 180,E1 11673.059,E2 11673.059} C_VEL
LIN {X 0,Y 497.697,Z 897.705,A -85,B 0,C 180,E1 11671.779,E2 11671.779} C_VEL
LIN {X 0,Y 494.379,Z 925.708,A -85,B 0,C 180,E1 11671.237,E2 11671.237} C_VEL
LIN {X 0,Y 490.182,Z 950.86,A -85,B 0,C 180,E1 11670.585,E2 11670.585} C_VEL
LIN {X 0,Y 485.959,Z 971.93,A -85,B 0,C 180,E1 11669.908,E2 11669.908} C_VEL
LIN {X 0,Y 481.193,Z 992.478,A -85,B 0,C 180,E1 11669.116,E2 11669.116} C_VEL
LIN {X 0,Y 475.294,Z 1014.886,A -85,B 0,C 180,E1 11668.089,E2 11668.089} C_VEL
LIN {X 0,Y 467.543,Z 1040.708,A -85,B 0,C 180,E1 11666.659,E2 11666.659} C_VEL
LIN {X 0,Y 460.742,Z 1060.866,A -85,B 0,C 180,E1 11665.338,E2 11665.338} C_VEL
LIN {X 0,Y 453.984,Z 1079.443,A -85,B 0,C 180,E1 11663.933,E2 11663.933} C_VEL
LIN {X 0,Y 446.905,Z 1097.688,A -85,B 0,C 180,E1 11662.352,E2 11662.352} C_VEL
LIN {X 0,Y 438.924,Z 1117.129,A -85,B 0,C 180,E1 11660.418,E2 11660.418} C_VEL
LIN {X 0,Y 429.477,Z 1138.667,A -85,B 0,C 180,E1 11657.893,E2 11657.893} C_VEL
LIN {X 0,Y 422.034,Z 1155.005,A -85,B 0,C 180,E1 11655.659,E2 11655.659} C_VEL
LIN {X 0,Y 415.075,Z 1169.976,A -85,B 0,C 180,E1 11653.322,E2 11653.322} C_VEL
LIN {X 0,Y 407.421,Z 1186.368,A -85,B 0,C 180,E1 11650.387,E2 11650.387} C_VEL
LIN {X 0,Y 400.003,Z 1202.131,A -85,B 0,C 180,E1 11647.047,E2 11647.047} C_VEL
LIN {X 0,Y 394.449,Z 1214.238,A -85,B 0,C 180,E1 11644.074,E2 11644.074} C_VEL
LIN {X 0,Y 389.744,Z 1224.99,A -85,B 0,C 180,E1 11641.045,E2 11641.045} C_VEL
LIN {X 0,Y 385.18,Z 1236.301,A -85,B 0,C 180,E1 11637.357,E2 11637.357} C_VEL
LIN {X 0,Y 381.433,Z 1246.497,A -85,B 0,C 180,E1 11633.321,E2 11633.321} C_VEL
LIN {X 0,Y 379.154,Z 1253.743,A -85,B 0,C 180,E1 11629.892,E2 11629.892} C_VEL
LIN {X 0,Y 377.676,Z 1259.52,A -85,B 0,C 180,E1 11626.618,E2 11626.618} C_VEL
LIN {X 0,Y 376.683,Z 1264.424,A -85,B 0,C 180,E1 11623.2,E2 11623.2} C_VEL
LIN {X 0,Y 376.114,Z 1268.665,A -85,B 0,C 180,E1 11619.337,E2 11619.337} C_VEL
LIN {X 0,Y 375.95,Z 1271.353,A -85,B 0,C 180,E1 11615.498,E2 11615.498} C_VEL
LIN {X 0,Y 375.912,Z 1272.573,A -85,B 0,C 180,E1 11612.138,E2 11612.138} C_VEL
LIN {X 0,Y 375.882,Z 1272.745,A -85,B 0,C 180,E1 11608.937,E2 11608.937} C_VEL
LIN {X 0,Y 375.927,Z 1272.003,A -85,B 0,C 180,E1 11605.886,E2 11605.886} C_VEL
LIN {X 0,Y 376.008,Z 1270.253,A -85,B 0,C 180,E1 11602.671,E2 11602.671} C_VEL
LIN {X 0,Y 376.237,Z 1267.506,A -85,B 0,C 180,E1 11599.439,E2 11599.439} C_VEL
LIN {X 0,Y 376.41,Z 1266.277,A -85,B 0,C 180,E1 11598.235,E2 11598.235} C_VEL
LIN {X 0,Y 375.63,Z 1265.046,A -85,B 0,C 180,E1 11597.074,E2 11597.074} C_VEL
LIN {X 0,Y 370.044,Z 1260.968,A -85,B 0,C 180,E1 11593.8,E2 11593.8} C_VEL
LIN {X 0,Y 369.796,Z 1259.669,A -85,B 0,C 180,E1 11592.96,E2 11592.96} C_VEL
LIN {X 0,Y 371.348,Z 1254.027,A -85,B 0,C 180,E1 11589.681,E2 11589.681} C_VEL
LIN {X 0,Y 373.616,Z 1247.163,A -85,B 0,C 180,E1 11586.338,E2 11586.338} C_VEL
LIN {X 0,Y 377.163,Z 1237.919,A -85,B 0,C 180,E1 11582.536,E2 11582.536} C_VEL
LIN {X 0,Y 382.244,Z 1225.903,A -85,B 0,C 180,E1 11578.462,E2 11578.462} C_VEL
LIN {X 0,Y 387.124,Z 1215.242,A -85,B 0,C 180,E1 11575.38,E2 11575.38} C_VEL
LIN {X 0,Y 392.561,Z 1203.864,A -85,B 0,C 180,E1 11572.508,E2 11572.508} C_VEL
LIN {X 0,Y 398.914,Z 1190.867,A -85,B 0,C 180,E1 11569.64,E2 11569.64} C_VEL
LIN {X 0,Y 407.713,Z 1172.92,A -85,B 0,C 180,E1 11566.252,E2 11566.252} C_VEL
LIN {X 0,Y 415.659,Z 1156.424,A -85,B 0,C 180,E1 11563.617,E2 11563.617} C_VEL
LIN {X 0,Y 423.046,Z 1140.775,A -85,B 0,C 180,E1 11561.437,E2 11561.437} C_VEL
LIN {X 0,Y 431.172,Z 1123.006,A -85,B 0,C 180,E1 11559.279,E2 11559.279} C_VEL
LIN {X 0,Y 440.97,Z 1100.285,A -85,B 0,C 180,E1 11556.933,E2 11556.933} C_VEL
LIN {X 0,Y 448.61,Z 1081.246,A -85,B 0,C 180,E1 11555.259,E2 11555.259} C_VEL
LIN {X 0,Y 455.483,Z 1062.967,A -85,B 0,C 180,E1 11553.861,E2 11553.861} C_VEL
LIN {X 0,Y 462.1,Z 1044.016,A -85,B 0,C 180,E1 11552.601,E2 11552.601} C_VEL
LIN {X 0,Y 469.019,Z 1022.216,A -85,B 0,C 180,E1 11551.344,E2 11551.344} C_VEL
LIN {X 0,Y 476.202,Z 996.523,A -85,B 0,C 180,E1 11550.119,E2 11550.119} C_VEL
LIN {X 0,Y 481.541,Z 974.352,A -85,B 0,C 180,E1 11549.247,E2 11549.247} C_VEL
LIN {X 0,Y 485.92,Z 953.349,A -85,B 0,C 180,E1 11548.563,E2 11548.563} C_VEL
LIN {X 0,Y 489.645,Z 932.002,A -85,B 0,C 180,E1 11547.991,E2 11547.991} C_VEL
LIN {X 0,Y 493.202,Z 906.483,A -85,B 0,C 180,E1 11547.456,E2 11547.456} C_VEL
LIN {X 0,Y 496.329,Z 868.694,A -85,B 0,C 180,E1 11546.834,E2 11546.834} C_VEL
LIN {X 0,Y 512.031,Z 649.185,A -85,B 0,C 180,E1 11543.418,E2 11543.418} C_VEL
LIN {X 0,Y 515.158,Z 605.866,A -85,B 0,C 180,E1 11542.721,E2 11542.721} C_VEL
LIN {X 0,Y 508.164,Z 594.998,A -85,B 0,C 180,E1 11540.322,E2 11540.322} C_VEL
LIN {X 0,Y 502.025,Z 585.961,A -85,B 0,C 180,E1 11537.922,E2 11537.922} C_VEL
LIN {X 0,Y 497.789,Z 579.887,A -85,B 0,C 180,E1 11536.033,E2 11536.033} C_VEL
LIN {X 0,Y 495.185,Z 576.2,A -85,B 0,C 180,E1 11534.739,E2 11534.739} C_VEL
LIN {X 0,Y 492.124,Z 571.793,A -85,B 0,C 180,E1 11533.034,E2 11533.034} C_VEL
LIN {X 0,Y 488.776,Z 567.086,A -85,B 0,C 180,E1 11530.848,E2 11530.848} C_VEL
LIN {X 0,Y 485.837,Z 563.112,A -85,B 0,C 180,E1 11528.462,E2 11528.462} C_VEL
LIN {X 0,Y 485.09,Z 561.793,A -85,B 0,C 180,E1 11527.7,E2 11527.7} C_VEL
LIN {X 0,Y 482.186,Z 558.206,A -85,B 0,C 180,E1 11523.686,E2 11523.686} C_VEL
LIN {X 0,Y 481.696,Z 556.104,A -85,B 0,C 180,E1 11521.784,E2 11521.784} C_VEL
LIN {X 0,Y 481.762,Z 556.353,A -85,B 0,C 180,E1 11517.978,E2 11517.978} C_VEL
LIN {X 0,Y 483.393,Z 560.323,A -85,B 0,C 180,E1 11514.302,E2 11514.302} C_VEL
LIN {X 0,Y 485.488,Z 562.352,A -85,B 0,C 180,E1 11512.009,E2 11512.009} C_VEL
LIN {X 0,Y 488.101,Z 566.47,A -85,B 0,C 180,E1 11509.734,E2 11509.734} C_VEL
LIN {X 0,Y 489.588,Z 568.176,A -85,B 0,C 180,E1 11508.693,E2 11508.693} C_VEL
LIN {X 0,Y 493.286,Z 573.469,A -85,B 0,C 180,E1 11506.401,E2 11506.401} C_VEL
LIN {X 0,Y 497.303,Z 579.173,A -85,B 0,C 180,E1 11504.31,E2 11504.31} C_VEL
LIN {X 0,Y 501.087,Z 584.666,A -85,B 0,C 180,E1 11502.583,E2 11502.583} C_VEL
LIN {X 0,Y 506.604,Z 592.703,A -85,B 0,C 180,E1 11500.365,E2 11500.365} C_VEL
LIN {X 0,Y 514.2,Z 605.55,A -85,B 0,C 180,E1 11497.656,E2 11497.656} C_VEL
LIN {X 0,Y 515.229,Z 607.606,A -85,B 0,C 180,E1 11497.307,E2 11497.307} C_VEL
LIN {X 0,Y 499.489,Z 825.307,A -85,B 0,C 180,E1 11493.921,E2 11493.921} C_VEL
LIN {X 0,Y 493.844,Z 902.935,A -85,B 0,C 180,E1 11492.692,E2 11492.692} C_VEL
LIN {X 0,Y 490.379,Z 931.239,A -85,B 0,C 180,E1 11492.149,E2 11492.149} C_VEL
LIN {X 0,Y 486.03,Z 956.386,A -85,B 0,C 180,E1 11491.513,E2 11491.513} C_VEL
LIN {X 0,Y 481.658,Z 977.544,A -85,B 0,C 180,E1 11490.844,E2 11490.844} C_VEL
LIN {X 0,Y 476.884,Z 997.536,A -85,B 0,C 180,E1 11490.087,E2 11490.087} C_VEL
LIN {X 0,Y 471.139,Z 1018.815,A -85,B 0,C 180,E1 11489.133,E2 11489.133} C_VEL
LIN {X 0,Y 463.347,Z 1044.382,A -85,B 0,C 180,E1 11487.76,E2 11487.76} C_VEL
LIN {X 0,Y 455.8,Z 1066.267,A -85,B 0,C 180,E1 11486.347,E2 11486.347} C_VEL
LIN {X 0,Y 448.627,Z 1085.54,A -85,B 0,C 180,E1 11484.898,E2 11484.898} C_VEL
LIN {X 0,Y 441.598,Z 1103.21,A -85,B 0,C 180,E1 11483.377,E2 11483.377} C_VEL
LIN {X 0,Y 433.886,Z 1121.517,A -85,B 0,C 180,E1 11481.575,E2 11481.575} C_VEL
LIN {X 0,Y 423.927,Z 1143.853,A -85,B 0,C 180,E1 11478.996,E2 11478.996} C_VEL
LIN {X 0,Y 416.094,Z 1160.624,A -85,B 0,C 180,E1 11476.72,E2 11476.72} C_VEL
LIN {X 0,Y 409.186,Z 1175.123,A -85,B 0,C 180,E1 11474.477,E2 11474.477} C_VEL
LIN {X 0,Y 402.457,Z 1189.077,A -85,B 0,C 180,E1 11472.025,E2 11472.025} C_VEL
LIN {X 0,Y 395.315,Z 1203.97,A -85,B 0,C 180,E1 11469.028,E2 11469.028} C_VEL
LIN {X 0,Y 388.114,Z 1219.181,A -85,B 0,C 180,E1 11465.42,E2 11465.42} C_VEL
LIN {X 0,Y 382.833,Z 1230.823,A -85,B 0,C 180,E1 11462.189,E2 11462.189} C_VEL
LIN {X 0,Y 378.646,Z 1240.617,A -85,B 0,C 180,E1 11459.064,E2 11459.064} C_VEL
LIN {X 0,Y 375.119,Z 1249.699,A -85,B 0,C 180,E1 11455.716,E2 11455.716} C_VEL
LIN {X 0,Y 371.821,Z 1259.421,A -85,B 0,C 180,E1 11451.446,E2 11451.446} C_VEL
LIN {X 0,Y 369.893,Z 1266.412,A -85,B 0,C 180,E1 11447.618,E2 11447.618} C_VEL
LIN {X 0,Y 368.832,Z 1271.39,A -85,B 0,C 180,E1 11444.277,E2 11444.277} C_VEL
LIN {X 0,Y 368.271,Z 1275.142,A -85,B 0,C 180,E1 11441.109,E2 11441.109} C_VEL
LIN {X 0,Y 367.987,Z 1277.947,A -85,B 0,C 180,E1 11437.961,E2 11437.961} C_VEL
LIN {X 0,Y 367.925,Z 1279.755,A -85,B 0,C 180,E1 11434.984,E2 11434.984} C_VEL
LIN {X 0,Y 367.91,Z 1280.76,A -85,B 0,C 180,E1 11431.864,E2 11431.864} C_VEL
LIN {X 0,Y 367.886,Z 1280.873,A -85,B 0,C 180,E1 11428.905,E2 11428.905} C_VEL
LIN {X 0,Y 367.919,Z 1280.094,A -85,B 0,C 180,E1 11425.788,E2 11425.788} C_VEL
LIN {X 0,Y 367.983,Z 1278.393,A -85,B 0,C 180,E1 11422.653,E2 11422.653} C_VEL
LIN {X 0,Y 368.207,Z 1275.612,A -85,B 0,C 180,E1 11419.355,E2 11419.355} C_VEL
LIN {X 0,Y 368.75,Z 1271.89,A -85,B 0,C 180,E1 11416.107,E2 11416.107} C_VEL
LIN {X 0,Y 369.71,Z 1267.162,A -85,B 0,C 180,E1 11412.851,E2 11412.851} C_VEL
LIN {X 0,Y 371.266,Z 1261.229,A -85,B 0,C 180,E1 11409.502,E2 11409.502} C_VEL
LIN {X 0,Y 373.783,Z 1253.45,A -85,B 0,C 180,E1 11405.837,E2 11405.837} C_VEL
LIN {X 0,Y 377.935,Z 1242.425,A -85,B 0,C 180,E1 11401.558,E2 11401.558} C_VEL
LIN {X 0,Y 382.2,Z 1232.236,A -85,B 0,C 180,E1 11398.239,E2 11398.239} C_VEL
LIN {X 0,Y 387.053,Z 1221.434,A -85,B 0,C 180,E1 11395.183,E2 11395.183} C_VEL
LIN {X 0,Y 392.774,Z 1209.173,A -85,B 0,C 180,E1 11392.153,E2 11392.153} C_VEL
LIN {X 0,Y 400.628,Z 1192.903,A -85,B 0,C 180,E1 11388.698,E2 11388.698} C_VEL
LIN {X 0,Y 408.482,Z 1176.51,A -85,B 0,C 180,E1 11385.76,E2 11385.76} C_VEL
LIN {X 0,Y 415.294,Z 1162.209,A -85,B 0,C 180,E1 11383.519,E2 11383.519} C_VEL
LIN {X 0,Y 422.5,Z 1146.771,A -85,B 0,C 180,E1 11381.388,E2 11381.388} C_VEL
LIN {X 0,Y 430.566,Z 1128.961,A -85,B 0,C 180,E1 11379.24,E2 11379.24} C_VEL
LIN {X 0,Y 440.525,Z 1105.688,A -85,B 0,C 180,E1 11376.859,E2 11376.859} C_VEL
LIN {X 0,Y 448,Z 1086.966,A -85,B 0,C 180,E1 11375.224,E2 11375.224} C_VEL
LIN {X 0,Y 454.928,Z 1068.453,A -85,B 0,C 180,E1 11373.816,E2 11373.816} C_VEL
LIN {X 0,Y 461.836,Z 1048.615,A -85,B 0,C 180,E1 11372.51,E2 11372.51} C_VEL
LIN {X 0,Y 469.302,Z 1025.073,A -85,B 0,C 180,E1 11371.18,E2 11371.18} C_VEL
LIN {X 0,Y 476.287,Z 999.558,A -85,B 0,C 180,E1 11370.003,E2 11370.003} C_VEL
LIN {X 0,Y 481.362,Z 978.459,A -85,B 0,C 180,E1 11369.195,E2 11369.195} C_VEL
LIN {X 0,Y 485.737,Z 957.416,A -85,B 0,C 180,E1 11368.523,E2 11368.523} C_VEL
LIN {X 0,Y 489.694,Z 934.774,A -85,B 0,C 180,E1 11367.94,E2 11367.94} C_VEL
LIN {X 0,Y 493.555,Z 905.033,A -85,B 0,C 180,E1 11367.349,E2 11367.349} C_VEL
LIN {X 0,Y 497.645,Z 850.228,A -85,B 0,C 180,E1 11366.475,E2 11366.475} C_VEL
LIN {X 0,Y 513.1,Z 634.528,A -85,B 0,C 180,E1 11363.115,E2 11363.115} C_VEL
LIN {X 0,Y 515.038,Z 607.204,A -85,B 0,C 180,E1 11362.667,E2 11362.667} C_VEL
LIN {X 0,Y 508.341,Z 595.719,A -85,B 0,C 180,E1 11360.344,E2 11360.344} C_VEL
LIN {X 0,Y 504.557,Z 589.777,A -85,B 0,C 180,E1 11358.906,E2 11358.906} C_VEL
LIN {X 0,Y 498.572,Z 581.047,A -85,B 0,C 180,E1 11356.366,E2 11356.366} C_VEL
LIN {X 0,Y 495.109,Z 576.172,A -85,B 0,C 180,E1 11354.682,E2 11354.682} C_VEL
LIN {X 0,Y 491.929,Z 571.613,A -85,B 0,C 180,E1 11352.92,E2 11352.92} C_VEL
LIN {X 0,Y 488.736,Z 567.078,A -85,B 0,C 180,E1 11350.849,E2 11350.849} C_VEL
LIN {X 0,Y 485.748,Z 563.065,A -85,B 0,C 180,E1 11348.464,E2 11348.464} C_VEL
LIN {X 0,Y 484.986,Z 561.73,A -85,B 0,C 180,E1 11347.701,E2 11347.701} C_VEL
LIN {X 0,Y 482.115,Z 558.24,A -85,B 0,C 180,E1 11343.924,E2 11343.924} C_VEL
LIN {X 0,Y 481.562,Z 556.064,A -85,B 0,C 180,E1 11342.142,E2 11342.142} C_VEL
LIN {X 0,Y 481.637,Z 556.244,A -85,B 0,C 180,E1 11337.382,E2 11337.382} C_VEL
LIN {X 0,Y 483.116,Z 560.004,A -85,B 0,C 180,E1 11334.179,E2 11334.179} C_VEL
LIN {X 0,Y 485.326,Z 562.157,A -85,B 0,C 180,E1 11331.768,E2 11331.768} C_VEL
LIN {X 0,Y 487.967,Z 566.291,A -85,B 0,C 180,E1 11329.492,E2 11329.492} C_VEL
LIN {X 0,Y 489.377,Z 567.924,A -85,B 0,C 180,E1 11328.509,E2 11328.509} C_VEL
LIN {X 0,Y 493.39,Z 573.655,A -85,B 0,C 180,E1 11326.045,E2 11326.045} C_VEL
LIN {X 0,Y 497.115,Z 578.899,A -85,B 0,C 180,E1 11324.124,E2 11324.124} C_VEL
LIN {X 0,Y 501.292,Z 584.979,A -85,B 0,C 180,E1 11322.231,E2 11322.231} C_VEL
LIN {X 0,Y 506.718,Z 592.914,A -85,B 0,C 180,E1 11320.069,E2 11320.069} C_VEL
LIN {X 0,Y 514.481,Z 604.815,A -85,B 0,C 180,E1 11317.368,E2 11317.368} C_VEL
LIN {X 0,Y 515.095,Z 606.184,A -85,B 0,C 180,E1 11317.155,E2 11317.155} C_VEL
LIN {X 0,Y 499.537,Z 821.201,A -85,B 0,C 180,E1 11313.81,E2 11313.81} C_VEL
LIN {X 0,Y 493.935,Z 898.03,A -85,B 0,C 180,E1 11312.596,E2 11312.596} C_VEL
LIN {X 0,Y 490.47,Z 926.392,A -85,B 0,C 180,E1 11312.045,E2 11312.045} C_VEL
LIN {X 0,Y 486.233,Z 951.199,A -85,B 0,C 180,E1 11311.405,E2 11311.405} C_VEL
LIN {X 0,Y 481.966,Z 972.028,A -85,B 0,C 180,E1 11310.737,E2 11310.737} C_VEL
LIN {X 0,Y 477.09,Z 992.576,A -85,B 0,C 180,E1 11309.95,E2 11309.95} C_VEL
LIN {X 0,Y 471.055,Z 1014.982,A -85,B 0,C 180,E1 11308.927,E2 11308.927} C_VEL
LIN {X 0,Y 462.882,Z 1041.47,A -85,B 0,C 180,E1 11307.461,E2 11307.461} C_VEL
LIN {X 0,Y 455.97,Z 1061.411,A -85,B 0,C 180,E1 11306.152,E2 11306.152} C_VEL
LIN {X 0,Y 448.914,Z 1080.27,A -85,B 0,C 180,E1 11304.721,E2 11304.721} C_VEL
LIN {X 0,Y 441.443,Z 1098.952,A -85,B 0,C 180,E1 11303.091,E2 11303.091} C_VEL
LIN {X 0,Y 432.178,Z 1120.719,A -85,B 0,C 180,E1 11300.884,E2 11300.884} C_VEL
LIN {X 0,Y 423.595,Z 1139.514,A -85,B 0,C 180,E1 11298.628,E2 11298.628} C_VEL
LIN {X 0,Y 416.318,Z 1154.968,A -85,B 0,C 180,E1 11296.499,E2 11296.499} C_VEL
LIN {X 0,Y 409.528,Z 1169.062,A -85,B 0,C 180,E1 11294.293,E2 11294.293} C_VEL
LIN {X 0,Y 402.533,Z 1183.399,A -85,B 0,C 180,E1 11291.74,E2 11291.74} C_VEL
LIN {X 0,Y 394.596,Z 1199.702,A -85,B 0,C 180,E1 11288.379,E2 11288.379} C_VEL
LIN {X 0,Y 387.847,Z 1213.71,A -85,B 0,C 180,E1 11284.933,E2 11284.933} C_VEL
LIN {X 0,Y 382.979,Z 1224.236,A -85,B 0,C 180,E1 11281.949,E2 11281.949} C_VEL
LIN {X 0,Y 378.726,Z 1233.985,A -85,B 0,C 180,E1 11278.773,E2 11278.773} C_VEL
LIN {X 0,Y 374.611,Z 1244.484,A -85,B 0,C 180,E1 11274.778,E2 11274.778} C_VEL
LIN {X 0,Y 371.573,Z 1253.235,A -85,B 0,C 180,E1 11270.645,E2 11270.645} C_VEL
LIN {X 0,Y 369.931,Z 1259.108,A -85,B 0,C 180,E1 11267.3,E2 11267.3} C_VEL
LIN {X 0,Y 368.872,Z 1263.901,A -85,B 0,C 180,E1 11263.964,E2 11263.964} C_VEL
LIN {X 0,Y 368.269,Z 1267.648,A -85,B 0,C 180,E1 11260.643,E2 11260.643} C_VEL
LIN {X 0,Y 368.008,Z 1270.491,A -85,B 0,C 180,E1 11257.184,E2 11257.184} C_VEL
LIN {X 0,Y 367.921,Z 1272.382,A -85,B 0,C 180,E1 11253.432,E2 11253.432} C_VEL
LIN {X 0,Y 367.88,Z 1272.922,A -85,B 0,C 180,E1 11249.537,E2 11249.537} C_VEL
LIN {X 0,Y 367.928,Z 1272.157,A -85,B 0,C 180,E1 11245.953,E2 11245.953} C_VEL
LIN {X 0,Y 368.011,Z 1270.418,A -85,B 0,C 180,E1 11242.619,E2 11242.619} C_VEL
LIN {X 0,Y 368.279,Z 1267.594,A -85,B 0,C 180,E1 11239.208,E2 11239.208} C_VEL
LIN {X 0,Y 368.853,Z 1264.031,A -85,B 0,C 180,E1 11236.042,E2 11236.042} C_VEL
LIN {X 0,Y 369.796,Z 1259.669,A -85,B 0,C 180,E1 11232.96,E2 11232.96} C_VEL
LIN {X 0,Y 369.259,Z 1257.924,A -85,B 0,C 180,E1 11231.791,E2 11231.791} C_VEL
LIN {X 0,Y 364.638,Z 1252.845,A -85,B 0,C 180,E1 11228.552,E2 11228.552} C_VEL
LIN {X 0,Y 364.641,Z 1251.151,A -85,B 0,C 180,E1 11227.628,E2 11227.628} C_VEL
LIN {X 0,Y 368.059,Z 1242.025,A -85,B 0,C 180,E1 11223.549,E2 11223.549} C_VEL
LIN {X 0,Y 371.849,Z 1233.124,A -85,B 0,C 180,E1 11220.175,E2 11220.175} C_VEL
LIN {X 0,Y 376.346,Z 1223.438,A -85,B 0,C 180,E1 11217.006,E2 11217.006} C_VEL
LIN {X 0,Y 382.254,Z 1211.348,A -85,B 0,C 180,E1 11213.582,E2 11213.582} C_VEL
LIN {X 0,Y 389.943,Z 1196.109,A -85,B 0,C 180,E1 11209.946,E2 11209.946} C_VEL
LIN {X 0,Y 396.924,Z 1182.377,A -85,B 0,C 180,E1 11207.144,E2 11207.144} C_VEL
LIN {X 0,Y 404.011,Z 1168.424,A -85,B 0,C 180,E1 11204.658,E2 11204.658} C_VEL
LIN {X 0,Y 411.585,Z 1153.264,A -85,B 0,C 180,E1 11202.294,E2 11202.294} C_VEL
LIN {X 0,Y 421.233,Z 1133.394,A -85,B 0,C 180,E1 11199.626,E2 11199.626} C_VEL
LIN {X 0,Y 430.292,Z 1113.528,A -85,B 0,C 180,E1 11197.381,E2 11197.381} C_VEL
LIN {X 0,Y 437.71,Z 1096.468,A -85,B 0,C 180,E1 11195.71,E2 11195.71} C_VEL
LIN {X 0,Y 445.005,Z 1078.62,A -85,B 0,C 180,E1 11194.176,E2 11194.176} C_VEL
LIN {X 0,Y 452.901,Z 1057.901,A -85,B 0,C 180,E1 11192.632,E2 11192.632} C_VEL
LIN {X 0,Y 461.74,Z 1032.078,A -85,B 0,C 180,E1 11191.023,E2 11191.023} C_VEL
LIN {X 0,Y 467.947,Z 1011.774,A -85,B 0,C 180,E1 11189.963,E2 11189.963} C_VEL
LIN {X 0,Y 473.497,Z 991.475,A -85,B 0,C 180,E1 11189.056,E2 11189.056} C_VEL
LIN {X 0,Y 478.492,Z 970.737,A -85,B 0,C 180,E1 11188.274,E2 11188.274} C_VEL
LIN {X 0,Y 483.463,Z 946.602,A -85,B 0,C 180,E1 11187.523,E2 11187.523} C_VEL
LIN {X 0,Y 487.991,Z 918.394,A -85,B 0,C 180,E1 11186.853,E2 11186.853} C_VEL
LIN {X 0,Y 490.665,Z 895.299,A -85,B 0,C 180,E1 11186.429,E2 11186.429} C_VEL
LIN {X 0,Y 506.205,Z 684.871,A -85,B 0,C 180,E1 11183.14,E2 11183.14} C_VEL
LIN {X 0,Y 511.738,Z 610.931,A -85,B 0,C 180,E1 11181.973,E2 11181.973} C_VEL
LIN {X 0,Y 504.018,Z 598.81,A -85,B 0,C 180,E1 11179.167,E2 11179.167} C_VEL
LIN {X 0,Y 497.16,Z 588.745,A -85,B 0,C 180,E1 11176.234,E2 11176.234} C_VEL
LIN {X 0,Y 493.768,Z 583.89,A -85,B 0,C 180,E1 11174.543,E2 11174.543} C_VEL
LIN {X 0,Y 490.661,Z 579.373,A -85,B 0,C 180,E1 11172.774,E2 11172.774} C_VEL
LIN {X 0,Y 487.472,Z 574.816,A -85,B 0,C 180,E1 11170.638,E2 11170.638} C_VEL
LIN {X 0,Y 484.558,Z 570.679,A -85,B 0,C 180,E1 11168.186,E2 11168.186} C_VEL
LIN {X 0,Y 483.998,Z 569.68,A -85,B 0,C 180,E1 11167.598,E2 11167.598} C_VEL
LIN {X 0,Y 481.158,Z 566.086,A -85,B 0,C 180,E1 11163.574,E2 11163.574} C_VEL
LIN {X 0,Y 480.693,Z 564.038,A -85,B 0,C 180,E1 11161.669,E2 11161.669} C_VEL
LIN {X 0,Y 480.76,Z 564.233,A -85,B 0,C 180,E1 11158.093,E2 11158.093} C_VEL
LIN {X 0,Y 482.331,Z 568.204,A -85,B 0,C 180,E1 11154.409,E2 11154.409} C_VEL
LIN {X 0,Y 484.329,Z 570.171,A -85,B 0,C 180,E1 11152.169,E2 11152.169} C_VEL
LIN {X 0,Y 486.97,Z 574.353,A -85,B 0,C 180,E1 11149.829,E2 11149.829} C_VEL
LIN {X 0,Y 488.351,Z 576.014,A -85,B 0,C 180,E1 11148.844,E2 11148.844} C_VEL
LIN {X 0,Y 491.994,Z 581.342,A -85,B 0,C 180,E1 11146.544,E2 11146.544} C_VEL
LIN {X 0,Y 495.85,Z 586.893,A -85,B 0,C 180,E1 11144.503,E2 11144.503} C_VEL
LIN {X 0,Y 501.184,Z 594.62,A -85,B 0,C 180,E1 11142.089,E2 11142.089} C_VEL
LIN {X 0,Y 505.799,Z 601.862,A -85,B 0,C 180,E1 11140.242,E2 11140.242} C_VEL
LIN {X 0,Y 511.81,Z 612.342,A -85,B 0,C 180,E1 11138.064,E2 11138.064} C_VEL
LIN {X 0,Y 495.731,Z 829.086,A -85,B 0,C 180,E1 11134.695,E2 11134.695} C_VEL
LIN {X 0,Y 490.19,Z 903.081,A -85,B 0,C 180,E1 11133.523,E2 11133.523} C_VEL
LIN {X 0,Y 486.583,Z 931.694,A -85,B 0,C 180,E1 11132.974,E2 11132.974} C_VEL
LIN {X 0,Y 482.215,Z 956.417,A -85,B 0,C 180,E1 11132.352,E2 11132.352} C_VEL
LIN {X 0,Y 477.787,Z 977.39,A -85,B 0,C 180,E1 11131.693,E2 11131.693} C_VEL
LIN {X 0,Y 472.926,Z 997.326,A -85,B 0,C 180,E1 11130.944,E2 11130.944} C_VEL
LIN {X 0,Y 467.014,Z 1018.733,A -85,B 0,C 180,E1 11129.99,E2 11129.99} C_VEL
LIN {X 0,Y 459.034,Z 1044.298,A -85,B 0,C 180,E1 11128.624,E2 11128.624} C_VEL
LIN {X 0,Y 451.302,Z 1066.182,A -85,B 0,C 180,E1 11127.214,E2 11127.214} C_VEL
LIN {X 0,Y 444.163,Z 1084.9,A -85,B 0,C 180,E1 11125.812,E2 11125.812} C_VEL
LIN {X 0,Y 436.989,Z 1102.454,A -85,B 0,C 180,E1 11124.31,E2 11124.31} C_VEL
LIN {X 0,Y 429.203,Z 1120.417,A -85,B 0,C 180,E1 11122.552,E2 11122.552} C_VEL
LIN {X 0,Y 419.485,Z 1141.745,A -85,B 0,C 180,E1 11120.119,E2 11120.119} C_VEL
LIN {X 0,Y 410.629,Z 1160.07,A -85,B 0,C 180,E1 11117.64,E2 11117.64} C_VEL
LIN {X 0,Y 403.341,Z 1174.827,A -85,B 0,C 180,E1 11115.347,E2 11115.347} C_VEL
LIN {X 0,Y 396.44,Z 1188.597,A -85,B 0,C 180,E1 11112.912,E2 11112.912} C_VEL
LIN {X 0,Y 389.452,Z 1202.582,A -85,B 0,C 180,E1 11110.084,E2 11110.084} C_VEL
LIN {X 0,Y 381.272,Z 1219.09,A -85,B 0,C 180,E1 11106.154,E2 11106.154} C_VEL
LIN {X 0,Y 375.748,Z 1230.732,A -85,B 0,C 180,E1 11102.871,E2 11102.871} C_VEL
LIN {X 0,Y 371.339,Z 1240.526,A -85,B 0,C 180,E1 11099.693,E2 11099.693} C_VEL
LIN {X 0,Y 367.642,Z 1249.537,A -85,B 0,C 180,E1 11096.309,E2 11096.309} C_VEL
LIN {X 0,Y 364.119,Z 1259.331,A -85,B 0,C 180,E1 11091.923,E2 11091.923} C_VEL
LIN {X 0,Y 362.053,Z 1266.323,A -85,B 0,C 180,E1 11088.012,E2 11088.012} C_VEL
LIN {X 0,Y 360.898,Z 1271.301,A -85,B 0,C 180,E1 11084.598,E2 11084.598} C_VEL
LIN {X 0,Y 360.299,Z 1275.053,A -85,B 0,C 180,E1 11081.359,E2 11081.359} C_VEL
LIN {X 0,Y 359.998,Z 1277.859,A -85,B 0,C 180,E1 11078.138,E2 11078.138} C_VEL
LIN {X 0,Y 359.927,Z 1279.668,A -85,B 0,C 180,E1 11075.095,E2 11075.095} C_VEL
LIN {X 0,Y 359.91,Z 1280.672,A -85,B 0,C 180,E1 11071.906,E2 11071.906} C_VEL
LIN {X 0,Y 359.887,Z 1280.785,A -85,B 0,C 180,E1 11068.881,E2 11068.881} C_VEL
LIN {X 0,Y 359.919,Z 1280.006,A -85,B 0,C 180,E1 11065.694,E2 11065.694} C_VEL
LIN {X 0,Y 359.979,Z 1278.309,A -85,B 0,C 180,E1 11062.494,E2 11062.494} C_VEL
LIN {X 0,Y 360.241,Z 1275.523,A -85,B 0,C 180,E1 11059.117,E2 11059.117} C_VEL
LIN {X 0,Y 360.799,Z 1271.909,A -85,B 0,C 180,E1 11055.881,E2 11055.881} C_VEL
LIN {X 0,Y 361.872,Z 1266.991,A -85,B 0,C 180,E1 11052.416,E2 11052.416} C_VEL
LIN {X 0,Y 363.507,Z 1261.137,A -85,B 0,C 180,E1 11049.044,E2 11049.044} C_VEL
LIN {X 0,Y 366.07,Z 1253.672,A -85,B 0,C 180,E1 11045.446,E2 11045.446} C_VEL
LIN {X 0,Y 370.576,Z 1242.332,A -85,B 0,C 180,E1 11040.94,E2 11040.94} C_VEL
LIN {X 0,Y 375.04,Z 1232.239,A -85,B 0,C 180,E1 11037.593,E2 11037.593} C_VEL
LIN {X 0,Y 380.171,Z 1221.34,A -85,B 0,C 180,E1 11034.458,E2 11034.458} C_VEL
LIN {X 0,Y 386.149,Z 1209.079,A -85,B 0,C 180,E1 11031.385,E2 11031.385} C_VEL
LIN {X 0,Y 394.187,Z 1193.148,A -85,B 0,C 180,E1 11027.956,E2 11027.956} C_VEL
LIN {X 0,Y 402.512,Z 1176.415,A -85,B 0,C 180,E1 11024.927,E2 11024.927} C_VEL
LIN {X 0,Y 409.667,Z 1161.931,A -85,B 0,C 180,E1 11022.643,E2 11022.643} C_VEL
LIN {X 0,Y 417.063,Z 1146.611,A -85,B 0,C 180,E1 11020.52,E2 11020.52} C_VEL
LIN {X 0,Y 425.448,Z 1128.669,A -85,B 0,C 180,E1 11018.35,E2 11018.35} C_VEL
LIN {X 0,Y 435.603,Z 1105.611,A -85,B 0,C 180,E1 11015.989,E2 11015.989} C_VEL
LIN {X 0,Y 443.297,Z 1086.871,A -85,B 0,C 180,E1 11014.354,E2 11014.354} C_VEL
LIN {X 0,Y 450.406,Z 1068.358,A -85,B 0,C 180,E1 11012.947,E2 11012.947} C_VEL
LIN {X 0,Y 457.537,Z 1048.363,A -85,B 0,C 180,E1 11011.634,E2 11011.634} C_VEL
LIN {X 0,Y 465.434,Z 1024.021,A -85,B 0,C 180,E1 11010.273,E2 11010.273} C_VEL
LIN {X 0,Y 472.394,Z 999.022,A -85,B 0,C 180,E1 11009.132,E2 11009.132} C_VEL
LIN {X 0,Y 477.468,Z 978.362,A -85,B 0,C 180,E1 11008.347,E2 11008.347} C_VEL
LIN {X 0,Y 481.946,Z 957.272,A -85,B 0,C 180,E1 11007.679,E2 11007.679} C_VEL
LIN {X 0,Y 485.998,Z 934.543,A -85,B 0,C 180,E1 11007.099,E2 11007.099} C_VEL
LIN {X 0,Y 489.969,Z 904.325,A -85,B 0,C 180,E1 11006.504,E2 11006.504} C_VEL
LIN {X 0,Y 494.472,Z 845.083,A -85,B 0,C 180,E1 11005.561,E2 11005.561} C_VEL
LIN {X 0,Y 510.369,Z 629.496,A -85,B 0,C 180,E1 11002.207,E2 11002.207} C_VEL
LIN {X 0,Y 511.629,Z 612.063,A -85,B 0,C 180,E1 11001.918,E2 11001.918} C_VEL
LIN {X 0,Y 504.195,Z 599.253,A -85,B 0,C 180,E1 10999.19,E2 10999.19} C_VEL
LIN {X 0,Y 497.468,Z 589.215,A -85,B 0,C 180,E1 10996.344,E2 10996.344} C_VEL
LIN {X 0,Y 493.471,Z 583.579,A -85,B 0,C 180,E1 10994.372,E2 10994.372} C_VEL
LIN {X 0,Y 490.464,Z 579.19,A -85,B 0,C 180,E1 10992.66,E2 10992.66} C_VEL
LIN {X 0,Y 487.428,Z 574.806,A -85,B 0,C 180,E1 10990.639,E2 10990.639} C_VEL
LIN {X 0,Y 484.463,Z 570.629,A -85,B 0,C 180,E1 10988.187,E2 10988.187} C_VEL
LIN {X 0,Y 483.768,Z 569.534,A -85,B 0,C 180,E1 10987.482,E2 10987.482} C_VEL
LIN {X 0,Y 481.031,Z 565.97,A -85,B 0,C 180,E1 10983.695,E2 10983.695} C_VEL
LIN {X 0,Y 480.55,Z 563.997,A -85,B 0,C 180,E1 10982.027,E2 10982.027} C_VEL
LIN {X 0,Y 480.626,Z 564.131,A -85,B 0,C 180,E1 10977.496,E2 10977.496} C_VEL
LIN {X 0,Y 482.14,Z 567.998,A -85,B 0,C 180,E1 10974.168,E2 10974.168} C_VEL
LIN {X 0,Y 484.219,Z 570.108,A -85,B 0,C 180,E1 10971.868,E2 10971.868} C_VEL
LIN {X 0,Y 486.995,Z 574.343,A -85,B 0,C 180,E1 10969.471,E2 10969.471} C_VEL
LIN {X 0,Y 488.219,Z 575.916,A -85,B 0,C 180,E1 10968.601,E2 10968.601} C_VEL
LIN {X 0,Y 491.897,Z 581.198,A -85,B 0,C 180,E1 10966.301,E2 10966.301} C_VEL
LIN {X 0,Y 495.661,Z 586.624,A -85,B 0,C 180,E1 10964.317,E2 10964.317} C_VEL
LIN {X 0,Y 501.228,Z 594.718,A -85,B 0,C 180,E1 10961.808,E2 10961.808} C_VEL
LIN {X 0,Y 507.694,Z 604.691,A -85,B 0,C 180,E1 10959.297,E2 10959.297} C_VEL
LIN {X 0,Y 511.661,Z 611.145,A -85,B 0,C 180,E1 10957.908,E2 10957.908} C_VEL
LIN {X 0,Y 495.699,Z 826.19,A -85,B 0,C 180,E1 10954.566,E2 10954.566} C_VEL
LIN {X 0,Y 490.276,Z 898.355,A -85,B 0,C 180,E1 10953.424,E2 10953.424} C_VEL
LIN {X 0,Y 486.668,Z 927.035,A -85,B 0,C 180,E1 10952.867,E2 10952.867} C_VEL
LIN {X 0,Y 482.397,Z 951.479,A -85,B 0,C 180,E1 10952.239,E2 10952.239} C_VEL
LIN {X 0,Y 478.076,Z 972.126,A -85,B 0,C 180,E1 10951.581,E2 10951.581} C_VEL
LIN {X 0,Y 473.092,Z 992.673,A -85,B 0,C 180,E1 10950.798,E2 10950.798} C_VEL
LIN {X 0,Y 466.968,Z 1014.906,A -85,B 0,C 180,E1 10949.788,E2 10949.788} C_VEL
LIN {X 0,Y 458.697,Z 1041.123,A -85,B 0,C 180,E1 10948.348,E2 10948.348} C_VEL
LIN {X 0,Y 451.628,Z 1061.057,A -85,B 0,C 180,E1 10947.047,E2 10947.047} C_VEL
LIN {X 0,Y 444.353,Z 1080.043,A -85,B 0,C 180,E1 10945.611,E2 10945.611} C_VEL
LIN {X 0,Y 437.107,Z 1097.717,A -85,B 0,C 180,E1 10944.077,E2 10944.077} C_VEL
LIN {X 0,Y 429.129,Z 1116.038,A -85,B 0,C 180,E1 10942.257,E2 10942.257} C_VEL
LIN {X 0,Y 419.016,Z 1137.867,A -85,B 0,C 180,E1 10939.708,E2 10939.708} C_VEL
LIN {X 0,Y 410.956,Z 1154.415,A -85,B 0,C 180,E1 10937.437,E2 10937.437} C_VEL
LIN {X 0,Y 403.592,Z 1169.157,A -85,B 0,C 180,E1 10935.121,E2 10935.121} C_VEL
LIN {X 0,Y 396.326,Z 1183.493,A -85,B 0,C 180,E1 10932.546,E2 10932.546} C_VEL
LIN {X 0,Y 388.045,Z 1199.826,A -85,B 0,C 180,E1 10929.14,E2 10929.14} C_VEL
LIN {X 0,Y 381.264,Z 1213.287,A -85,B 0,C 180,E1 10925.794,E2 10925.794} C_VEL
LIN {X 0,Y 375.989,Z 1224.156,A -85,B 0,C 180,E1 10922.677,E2 10922.677} C_VEL
LIN {X 0,Y 371.557,Z 1233.758,A -85,B 0,C 180,E1 10919.506,E2 10919.506} C_VEL
LIN {X 0,Y 367.519,Z 1243.38,A -85,B 0,C 180,E1 10915.808,E2 10915.808} C_VEL
LIN {X 0,Y 364.014,Z 1252.819,A -85,B 0,C 180,E1 10911.379,E2 10911.379} C_VEL
LIN {X 0,Y 362.163,Z 1258.947,A -85,B 0,C 180,E1 10907.85,E2 10907.85} C_VEL
LIN {X 0,Y 360.988,Z 1263.787,A -85,B 0,C 180,E1 10904.439,E2 10904.439} C_VEL
LIN {X 0,Y 360.358,Z 1267.422,A -85,B 0,C 180,E1 10901.204,E2 10901.204} C_VEL
LIN {X 0,Y 360.017,Z 1270.243,A -85,B 0,C 180,E1 10897.826,E2 10897.826} C_VEL
LIN {X 0,Y 359.933,Z 1271.932,A -85,B 0,C 180,E1 10894.785,E2 10894.785} C_VEL
LIN {X 0,Y 359.91,Z 1272.815,A -85,B 0,C 180,E1 10891.756,E2 10891.756} C_VEL
LIN {X 0,Y 359.892,Z 1272.897,A -85,B 0,C 180,E1 10888.731,E2 10888.731} C_VEL
LIN {X 0,Y 359.93,Z 1272.11,A -85,B 0,C 180,E1 10885.544,E2 10885.544} C_VEL
LIN {X 0,Y 360.016,Z 1270.429,A -85,B 0,C 180,E1 10882.344,E2 10882.344} C_VEL
LIN {X 0,Y 360.319,Z 1267.682,A -85,B 0,C 180,E1 10878.966,E2 10878.966} C_VEL
LIN {X 0,Y 360.932,Z 1264.122,A -85,B 0,C 180,E1 10875.732,E2 10875.732} C_VEL
LIN {X 0,Y 362.048,Z 1259.359,A -85,B 0,C 180,E1 10872.32,E2 10872.32} C_VEL
LIN {X 0,Y 363.785,Z 1253.517,A -85,B 0,C 180,E1 10868.902,E2 10868.902} C_VEL
LIN {X 0,Y 364.641,Z 1251.151,A -85,B 0,C 180,E1 10867.628,E2 10867.628} C_VEL
LIN {X 0,Y 364.532,Z 1248.922,A -85,B 0,C 180,E1 10866.46,E2 10866.46} C_VEL
LIN {X 0,Y 361.052,Z 1242.785,A -85,B 0,C 180,E1 10863.291,E2 10863.291} C_VEL
LIN {X 0,Y 361.326,Z 1240.495,A -85,B 0,C 180,E1 10862.297,E2 10862.297} C_VEL
LIN {X 0,Y 365.736,Z 1230.938,A -85,B 0,C 180,E1 10858.712,E2 10858.712} C_VEL
LIN {X 0,Y 372.59,Z 1217.129,A -85,B 0,C 180,E1 10854.392,E2 10854.392} C_VEL
LIN {X 0,Y 378.715,Z 1205.304,A -85,B 0,C 180,E1 10851.272,E2 10851.272} C_VEL
LIN {X 0,Y 385.015,Z 1193.414,A -85,B 0,C 180,E1 10848.537,E2 10848.537} C_VEL
LIN {X 0,Y 392.022,Z 1180.202,A -85,B 0,C 180,E1 10845.877,E2 10845.877} C_VEL
LIN {X 0,Y 401.107,Z 1163.007,A -85,B 0,C 180,E1 10842.88,E2 10842.88} C_VEL
LIN {X 0,Y 410.611,Z 1144.209,A -85,B 0,C 180,E1 10840.136,E2 10840.136} C_VEL
LIN {X 0,Y 418.818,Z 1127.428,A -85,B 0,C 180,E1 10838.025,E2 10838.025} C_VEL
LIN {X 0,Y 426.575,Z 1110.844,A -85,B 0,C 180,E1 10836.206,E2 10836.206} C_VEL
LIN {X 0,Y 435.269,Z 1091.231,A -85,B 0,C 180,E1 10834.338,E2 10834.338} C_VEL
LIN {X 0,Y 445.145,Z 1066.886,A -85,B 0,C 180,E1 10832.385,E2 10832.385} C_VEL
LIN {X 0,Y 452.322,Z 1047.564,A -85,B 0,C 180,E1 10831.075,E2 10831.075} C_VEL
LIN {X 0,Y 458.856,Z 1028.249,A -85,B 0,C 180,E1 10829.935,E2 10829.935} C_VEL
LIN {X 0,Y 464.939,Z 1008.471,A -85,B 0,C 180,E1 10828.934,E2 10828.934} C_VEL
LIN {X 0,Y 471.044,Z 986.196,A -85,B 0,C 180,E1 10827.977,E2 10827.977} C_VEL
LIN {X 0,Y 477.526,Z 958.052,A -85,B 0,C 180,E1 10827.004,E2 10827.004} C_VEL
LIN {X 0,Y 481.759,Z 935.453,A -85,B 0,C 180,E1 10826.385,E2 10826.385} C_VEL
LIN {X 0,Y 485.054,Z 913.728,A -85,B 0,C 180,E1 10825.914,E2 10825.914} C_VEL
LIN {X 0,Y 487.618,Z 890.294,A -85,B 0,C 180,E1 10825.498,E2 10825.498} C_VEL
LIN {X 0,Y 504.06,Z 672.574,A -85,B 0,C 180,E1 10822.109,E2 10822.109} C_VEL
LIN {X 0,Y 508.392,Z 616.125,A -85,B 0,C 180,E1 10821.216,E2 10821.216} C_VEL
LIN {X 0,Y 501.91,Z 605.796,A -85,B 0,C 180,E1 10818.768,E2 10818.768} C_VEL
LIN {X 0,Y 495.579,Z 596.289,A -85,B 0,C 180,E1 10815.986,E2 10815.986} C_VEL
LIN {X 0,Y 492.144,Z 591.3,A -85,B 0,C 180,E1 10814.231,E2 10814.231} C_VEL
LIN {X 0,Y 489.208,Z 586.951,A -85,B 0,C 180,E1 10812.513,E2 10812.513} C_VEL
LIN {X 0,Y 486.338,Z 582.697,A -85,B 0,C 180,E1 10810.543,E2 10810.543} C_VEL
LIN {X 0,Y 483.399,Z 578.49,A -85,B 0,C 180,E1 10808.026,E2 10808.026} C_VEL
LIN {X 0,Y 482.789,Z 577.488,A -85,B 0,C 180,E1 10807.378,E2 10807.378} C_VEL
LIN {X 0,Y 480.132,Z 573.965,A -85,B 0,C 180,E1 10803.462,E2 10803.462} C_VEL
LIN {X 0,Y 479.692,Z 571.972,A -85,B 0,C 180,E1 10801.553,E2 10801.553} C_VEL
LIN {X 0,Y 479.774,Z 572.263,A -85,B 0,C 180,E1 10798.089,E2 10798.089} C_VEL
LIN {X 0,Y 481.356,Z 576.183,A -85,B 0,C 180,E1 10794.397,E2 10794.397} C_VEL
LIN {X 0,Y 483.175,Z 577.988,A -85,B 0,C 180,E1 10792.329,E2 10792.329} C_VEL
LIN {X 0,Y 485.841,Z 582.237,A -85,B 0,C 180,E1 10789.925,E2 10789.925} C_VEL
LIN {X 0,Y 487.117,Z 583.849,A -85,B 0,C 180,E1 10788.995,E2 10788.995} C_VEL
LIN {X 0,Y 490.514,Z 588.884,A -85,B 0,C 180,E1 10786.803,E2 10786.803} C_VEL
LIN {X 0,Y 494.404,Z 594.61,A -85,B 0,C 180,E1 10784.697,E2 10784.697} C_VEL
LIN {X 0,Y 499.494,Z 602.137,A -85,B 0,C 180,E1 10782.346,E2 10782.346} C_VEL
LIN {X 0,Y 503.935,Z 609.246,A -85,B 0,C 180,E1 10780.528,E2 10780.528} C_VEL
LIN {X 0,Y 508.458,Z 617.375,A -85,B 0,C 180,E1 10778.826,E2 10778.826} C_VEL
LIN {X 0,Y 492.078,Z 832.691,A -85,B 0,C 180,E1 10775.483,E2 10775.483} C_VEL
LIN {X 0,Y 486.64,Z 903.228,A -85,B 0,C 180,E1 10774.367,E2 10774.367} C_VEL
LIN {X 0,Y 482.86,Z 932.327,A -85,B 0,C 180,E1 10773.807,E2 10773.807} C_VEL
LIN {X 0,Y 478.506,Z 956.447,A -85,B 0,C 180,E1 10773.204,E2 10773.204} C_VEL
LIN {X 0,Y 474.006,Z 977.31,A -85,B 0,C 180,E1 10772.554,E2 10772.554} C_VEL
LIN {X 0,Y 469.042,Z 997.245,A -85,B 0,C 180,E1 10771.81,E2 10771.81} C_VEL
LIN {X 0,Y 463.327,Z 1017.518,A -85,B 0,C 180,E1 10770.916,E2 10770.916} C_VEL
LIN {X 0,Y 455.48,Z 1042.403,A -85,B 0,C 180,E1 10769.613,E2 10769.613} C_VEL
LIN {X 0,Y 446.943,Z 1066.015,A -85,B 0,C 180,E1 10768.105,E2 10768.105} C_VEL
LIN {X 0,Y 439.588,Z 1084.814,A -85,B 0,C 180,E1 10766.7,E2 10766.7} C_VEL
LIN {X 0,Y 432.21,Z 1102.367,A -85,B 0,C 180,E1 10765.201,E2 10765.201} C_VEL
LIN {X 0,Y 424.018,Z 1120.732,A -85,B 0,C 180,E1 10763.402,E2 10763.402} C_VEL
LIN {X 0,Y 413.674,Z 1142.658,A -85,B 0,C 180,E1 10760.876,E2 10760.876} C_VEL
LIN {X 0,Y 405.03,Z 1159.981,A -85,B 0,C 180,E1 10758.516,E2 10758.516} C_VEL
LIN {X 0,Y 397.481,Z 1174.738,A -85,B 0,C 180,E1 10756.208,E2 10756.208} C_VEL
LIN {X 0,Y 390.288,Z 1188.57,A -85,B 0,C 180,E1 10753.741,E2 10753.741} C_VEL
LIN {X 0,Y 382.749,Z 1203.086,A -85,B 0,C 180,E1 10750.767,E2 10750.767} C_VEL
LIN {X 0,Y 374.502,Z 1218.999,A -85,B 0,C 180,E1 10746.915,E2 10746.915} C_VEL
LIN {X 0,Y 368.702,Z 1230.641,A -85,B 0,C 180,E1 10743.582,E2 10743.582} C_VEL
LIN {X 0,Y 364.08,Z 1240.436,A -85,B 0,C 180,E1 10740.346,E2 10740.346} C_VEL
LIN {X 0,Y 360.007,Z 1249.855,A -85,B 0,C 180,E1 10736.733,E2 10736.733} C_VEL
LIN {X 0,Y 356.204,Z 1259.853,A -85,B 0,C 180,E1 10732.089,E2 10732.089} C_VEL
LIN {X 0,Y 354.149,Z 1266.49,A -85,B 0,C 180,E1 10728.258,E2 10728.258} C_VEL
LIN {X 0,Y 352.974,Z 1271.212,A -85,B 0,C 180,E1 10724.933,E2 10724.933} C_VEL
LIN {X 0,Y 352.331,Z 1274.965,A -85,B 0,C 180,E1 10721.619,E2 10721.619} C_VEL
LIN {X 0,Y 352.01,Z 1277.771,A -85,B 0,C 180,E1 10718.324,E2 10718.324} C_VEL
LIN {X 0,Y 351.928,Z 1279.58,A -85,B 0,C 180,E1 10715.211,E2 10715.211} C_VEL
LIN {X 0,Y 351.911,Z 1280.585,A -85,B 0,C 180,E1 10711.949,E2 10711.949} C_VEL
LIN {X 0,Y 351.888,Z 1280.697,A -85,B 0,C 180,E1 10708.856,E2 10708.856} C_VEL
LIN {X 0,Y 351.92,Z 1279.918,A -85,B 0,C 180,E1 10705.596,E2 10705.596} C_VEL
LIN {X 0,Y 351.98,Z 1278.22,A -85,B 0,C 180,E1 10702.323,E2 10702.323} C_VEL
LIN {X 0,Y 352.272,Z 1275.434,A -85,B 0,C 180,E1 10698.867,E2 10698.867} C_VEL
LIN {X 0,Y 352.867,Z 1271.819,A -85,B 0,C 180,E1 10695.556,E2 10695.556} C_VEL
LIN {X 0,Y 354.011,Z 1266.98,A -85,B 0,C 180,E1 10692.065,E2 10692.065} C_VEL
LIN {X 0,Y 355.775,Z 1261.046,A -85,B 0,C 180,E1 10688.566,E2 10688.566} C_VEL
LIN {X 0,Y 358.479,Z 1253.622,A -85,B 0,C 180,E1 10684.911,E2 10684.911} C_VEL
LIN {X 0,Y 363.267,Z 1242.239,A -85,B 0,C 180,E1 10680.297,E2 10680.297} C_VEL
LIN {X 0,Y 368.221,Z 1231.627,A -85,B 0,C 180,E1 10676.731,E2 10676.731} C_VEL
LIN {X 0,Y 373.341,Z 1221.246,A -85,B 0,C 180,E1 10673.706,E2 10673.706} C_VEL
LIN {X 0,Y 379.602,Z 1208.985,A -85,B 0,C 180,E1 10670.591,E2 10670.591} C_VEL
LIN {X 0,Y 388.319,Z 1192.375,A -85,B 0,C 180,E1 10666.994,E2 10666.994} C_VEL
LIN {X 0,Y 396.628,Z 1176.321,A -85,B 0,C 180,E1 10664.068,E2 10664.068} C_VEL
LIN {X 0,Y 403.868,Z 1162.177,A -85,B 0,C 180,E1 10661.82,E2 10661.82} C_VEL
LIN {X 0,Y 411.265,Z 1147.372,A -85,B 0,C 180,E1 10659.749,E2 10659.749} C_VEL
LIN {X 0,Y 419.125,Z 1131.074,A -85,B 0,C 180,E1 10657.747,E2 10657.747} C_VEL
LIN {X 0,Y 428.806,Z 1110.158,A -85,B 0,C 180,E1 10655.529,E2 10655.529} C_VEL
LIN {X 0,Y 438.099,Z 1088.251,A -85,B 0,C 180,E1 10653.584,E2 10653.584} C_VEL
LIN {X 0,Y 445.657,Z 1069.141,A -85,B 0,C 180,E1 10652.123,E2 10652.123} C_VEL
LIN {X 0,Y 452.602,Z 1050.23,A -85,B 0,C 180,E1 10650.874,E2 10650.874} C_VEL
LIN {X 0,Y 459.384,Z 1030.004,A -85,B 0,C 180,E1 10649.718,E2 10649.718} C_VEL
LIN {X 0,Y 467.043,Z 1004.516,A -85,B 0,C 180,E1 10648.495,E2 10648.495} C_VEL
LIN {X 0,Y 473.123,Z 980.677,A -85,B 0,C 180,E1 10647.57,E2 10647.57} C_VEL
LIN {X 0,Y 477.915,Z 958.849,A -85,B 0,C 180,E1 10646.872,E2 10646.872} C_VEL
LIN {X 0,Y 481.871,Z 937.457,A -85,B 0,C 180,E1 10646.317,E2 10646.317} C_VEL
LIN {X 0,Y 485.396,Z 913.496,A -85,B 0,C 180,E1 10645.823,E2 10645.823} C_VEL
